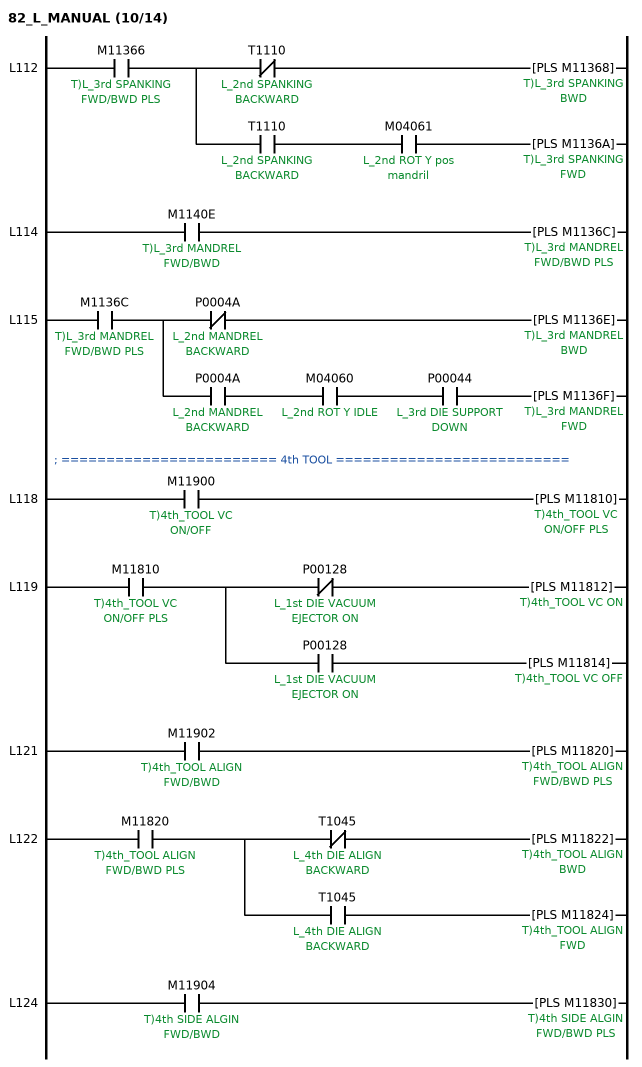
[picture p336: 82_L_MANUAL rungs L112-L124]
; L112
LOAD      M11366	// T)L_3rd SPANKING FWD/BWD PLS
MPUSH
AND NOT   T1110	// L_2nd SPANKING BACKWARD
OUTP      M11368	// T)L_3rd SPANKING BWD
MPOP
AND       T1110	// L_2nd SPANKING BACKWARD
AND       M04061	// L_2nd ROT Y pos mandril
OUTP      M1136A	// T)L_3rd SPANKING FWD
; L114
LOAD      M1140E	// T)L_3rd MANDREL FWD/BWD
OUTP      M1136C	// T)L_3rd MANDREL FWD/BWD PLS
; L115
LOAD      M1136C	// T)L_3rd MANDREL FWD/BWD PLS
MPUSH
AND NOT   P0004A	// L_2nd MANDREL BACKWARD
OUTP      M1136E	// T)L_3rd MANDREL BWD
MPOP
AND       P0004A	// L_2nd MANDREL BACKWARD
AND       M04060	// L_2nd ROT Y IDLE
AND       P00044	// L_3rd DIE SUPPORT DOWN
OUTP      M1136F	// T)L_3rd MANDREL FWD
// ======================== 4th TOOL ==========================
; L118
LOAD      M11900	// T)4th_TOOL VC ON/OFF
OUTP      M11810	// T)4th_TOOL VC ON/OFF PLS
; L119
LOAD      M11810	// T)4th_TOOL VC ON/OFF PLS
MPUSH
AND NOT   P00128	// L_1st DIE VACUUM EJECTOR ON
OUTP      M11812	// T)4th_TOOL VC ON
MPOP
AND       P00128	// L_1st DIE VACUUM EJECTOR ON
OUTP      M11814	// T)4th_TOOL VC OFF
; L121
LOAD      M11902	// T)4th_TOOL ALIGN FWD/BWD
OUTP      M11820	// T)4th_TOOL ALIGN FWD/BWD PLS
; L122
LOAD      M11820	// T)4th_TOOL ALIGN FWD/BWD PLS
MPUSH
AND NOT   T1045	// L_4th DIE ALIGN BACKWARD
OUTP      M11822	// T)4th_TOOL ALIGN BWD
MPOP
AND       T1045	// L_4th DIE ALIGN BACKWARD
OUTP      M11824	// T)4th_TOOL ALIGN FWD
; L124
LOAD      M11904	// T)4th SIDE ALGIN FWD/BWD
OUTP      M11830	// T)4th SIDE ALGIN FWD/BWD PLS

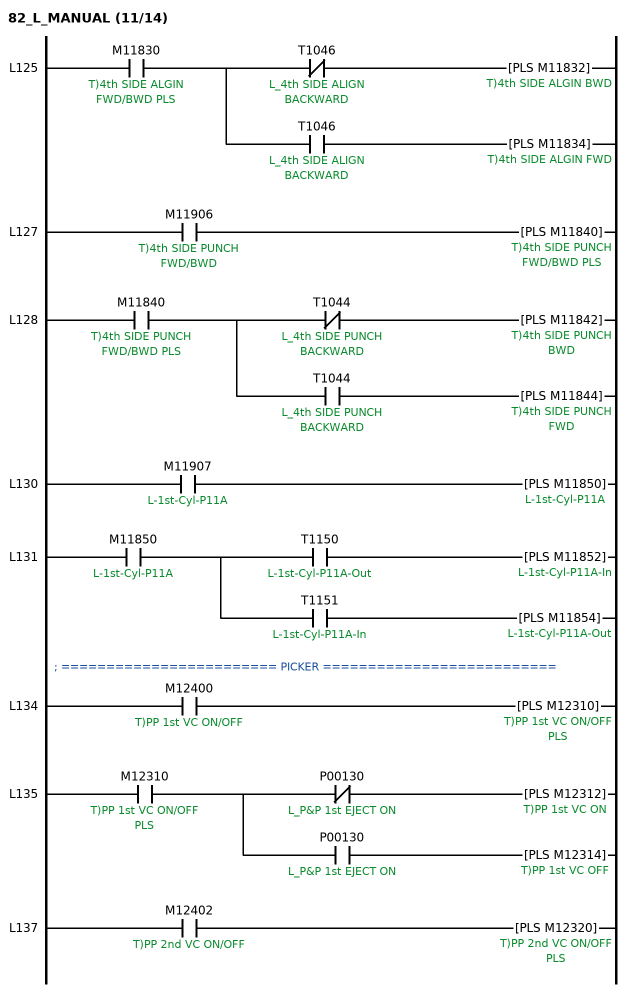
; L125
LOAD      M11830	// T)4th SIDE ALGIN FWD/BWD PLS
MPUSH
AND NOT   T1046	// L_4th SIDE ALIGN BACKWARD
OUTP      M11832	// T)4th SIDE ALGIN BWD
MPOP
AND       T1046	// L_4th SIDE ALIGN BACKWARD
OUTP      M11834	// T)4th SIDE ALGIN FWD
; L127
LOAD      M11906	// T)4th SIDE PUNCH FWD/BWD
OUTP      M11840	// T)4th SIDE PUNCH FWD/BWD PLS
; L128
LOAD      M11840	// T)4th SIDE PUNCH FWD/BWD PLS
MPUSH
AND NOT   T1044	// L_4th SIDE PUNCH BACKWARD
OUTP      M11842	// T)4th SIDE PUNCH BWD
MPOP
AND       T1044	// L_4th SIDE PUNCH BACKWARD
OUTP      M11844	// T)4th SIDE PUNCH FWD
; L130
LOAD      M11907	// L-1st-Cyl-P11A
OUTP      M11850	// L-1st-Cyl-P11A
; L131
LOAD      M11850	// L-1st-Cyl-P11A
MPUSH
AND       T1150	// L-1st-Cyl-P11A-Out
OUTP      M11852	// L-1st-Cyl-P11A-In
MPOP
AND       T1151	// L-1st-Cyl-P11A-In
OUTP      M11854	// L-1st-Cyl-P11A-Out
// ======================== PICKER ==========================
; L134
LOAD      M12400	// T)PP 1st VC ON/OFF
OUTP      M12310	// T)PP 1st VC ON/OFF PLS
; L135
LOAD      M12310	// T)PP 1st VC ON/OFF PLS
MPUSH
AND NOT   P00130	// L_P&P 1st EJECT ON
OUTP      M12312	// T)PP 1st VC ON
MPOP
AND       P00130	// L_P&P 1st EJECT ON
OUTP      M12314	// T)PP 1st VC OFF
; L137
LOAD      M12402	// T)PP 2nd VC ON/OFF
OUTP      M12320	// T)PP 2nd VC ON/OFF PLS

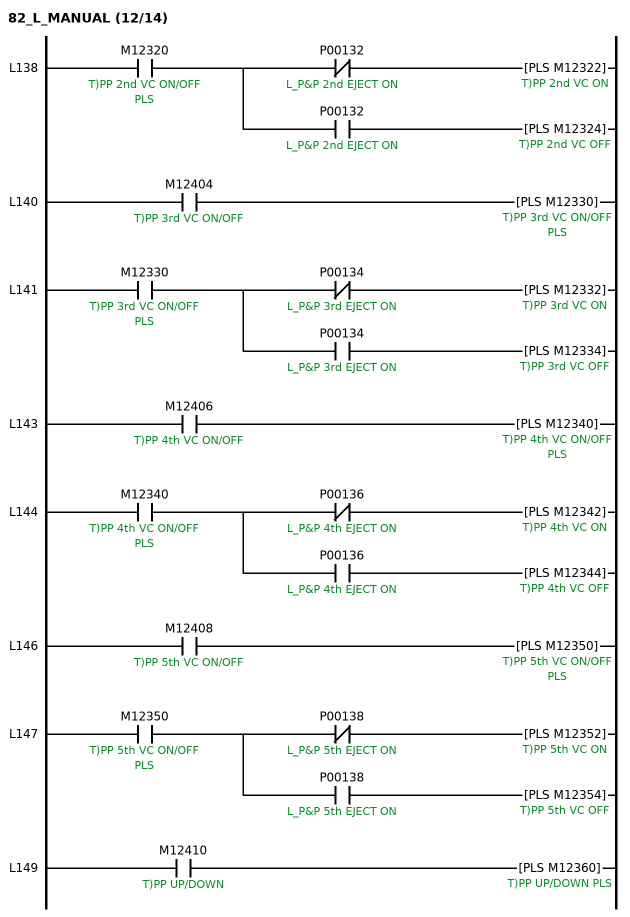
; L138
LOAD      M12320	// T)PP 2nd VC ON/OFF PLS
MPUSH
AND NOT   P00132	// L_P&P 2nd EJECT ON
OUTP      M12322	// T)PP 2nd VC ON
MPOP
AND       P00132	// L_P&P 2nd EJECT ON
OUTP      M12324	// T)PP 2nd VC OFF
; L140
LOAD      M12404	// T)PP 3rd VC ON/OFF
OUTP      M12330	// T)PP 3rd VC ON/OFF PLS
; L141
LOAD      M12330	// T)PP 3rd VC ON/OFF PLS
MPUSH
AND NOT   P00134	// L_P&P 3rd EJECT ON
OUTP      M12332	// T)PP 3rd VC ON
MPOP
AND       P00134	// L_P&P 3rd EJECT ON
OUTP      M12334	// T)PP 3rd VC OFF
; L143
LOAD      M12406	// T)PP 4th VC ON/OFF
OUTP      M12340	// T)PP 4th VC ON/OFF PLS
; L144
LOAD      M12340	// T)PP 4th VC ON/OFF PLS
MPUSH
AND NOT   P00136	// L_P&P 4th EJECT ON
OUTP      M12342	// T)PP 4th VC ON
MPOP
AND       P00136	// L_P&P 4th EJECT ON
OUTP      M12344	// T)PP 4th VC OFF
; L146
LOAD      M12408	// T)PP 5th VC ON/OFF
OUTP      M12350	// T)PP 5th VC ON/OFF PLS
; L147
LOAD      M12350	// T)PP 5th VC ON/OFF PLS
MPUSH
AND NOT   P00138	// L_P&P 5th EJECT ON
OUTP      M12352	// T)PP 5th VC ON
MPOP
AND       P00138	// L_P&P 5th EJECT ON
OUTP      M12354	// T)PP 5th VC OFF
; L149
LOAD      M12410	// T)PP UP/DOWN
OUTP      M12360	// T)PP UP/DOWN PLS

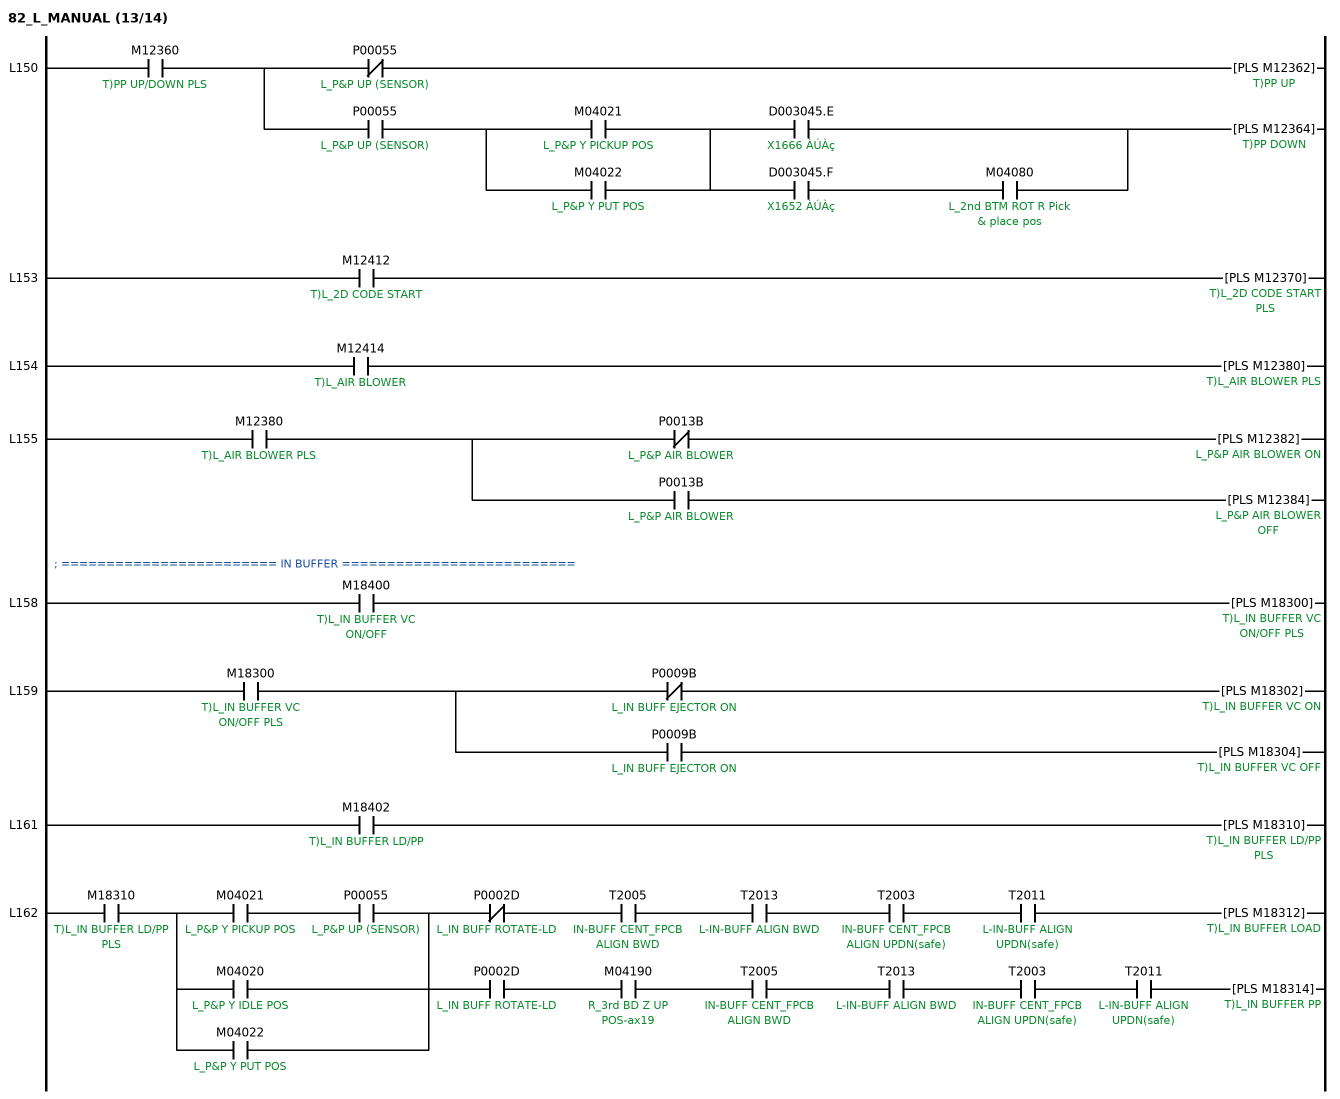
; L150
LOAD      M12360	// T)PP UP/DOWN PLS
MPUSH
AND NOT   P00055	// L_P&P UP (SENSOR)
OUTP      M12362	// T)PP UP
MPOP
AND       P00055	// L_P&P UP (SENSOR)
LOAD      M04021	// L_P&P Y PICKUP POS
OR        M04022	// L_P&P Y PUT POS
AND LOAD
LOAD      D003045.E	// X1666 ÀÚÀç
LOAD      D003045.F	// X1652 ÀÚÀç
AND       M04080	// L_2nd BTM ROT R Pick & place pos
OR LOAD
AND LOAD
OUTP      M12364	// T)PP DOWN
; L153
LOAD      M12412	// T)L_2D CODE START
OUTP      M12370	// T)L_2D CODE START PLS
; L154
LOAD      M12414	// T)L_AIR BLOWER
OUTP      M12380	// T)L_AIR BLOWER PLS
; L155
LOAD      M12380	// T)L_AIR BLOWER PLS
MPUSH
AND NOT   P0013B	// L_P&P AIR BLOWER
OUTP      M12382	// L_P&P AIR BLOWER ON
MPOP
AND       P0013B	// L_P&P AIR BLOWER
OUTP      M12384	// L_P&P AIR BLOWER OFF
// ======================== IN BUFFER ==========================
; L158
LOAD      M18400	// T)L_IN BUFFER VC ON/OFF
OUTP      M18300	// T)L_IN BUFFER VC ON/OFF PLS
; L159
LOAD      M18300	// T)L_IN BUFFER VC ON/OFF PLS
MPUSH
AND NOT   P0009B	// L_IN BUFF EJECTOR ON
OUTP      M18302	// T)L_IN BUFFER VC ON
MPOP
AND       P0009B	// L_IN BUFF EJECTOR ON
OUTP      M18304	// T)L_IN BUFFER VC OFF
; L161
LOAD      M18402	// T)L_IN BUFFER LD/PP
OUTP      M18310	// T)L_IN BUFFER LD/PP PLS
; L162
LOAD      M18310	// T)L_IN BUFFER LD/PP PLS
LOAD      M04021	// L_P&P Y PICKUP POS
AND       P00055	// L_P&P UP (SENSOR)
OR        M04020	// L_P&P Y IDLE POS
OR        M04022	// L_P&P Y PUT POS
AND LOAD
MPUSH
AND NOT   P0002D	// L_IN BUFF ROTATE-LD
AND       T2005	// IN-BUFF CENT_FPCB ALIGN BWD
AND       T2013	// L-IN-BUFF ALIGN BWD
AND       T2003	// IN-BUFF CENT_FPCB ALIGN UPDN(safe)
AND       T2011	// L-IN-BUFF ALIGN UPDN(safe)
OUTP      M18312	// T)L_IN BUFFER LOAD
MPOP
AND       P0002D	// L_IN BUFF ROTATE-LD
AND       M04190	// R_3rd BD Z UP POS-ax19
AND       T2005	// IN-BUFF CENT_FPCB ALIGN BWD
AND       T2013	// L-IN-BUFF ALIGN BWD
AND       T2003	// IN-BUFF CENT_FPCB ALIGN UPDN(safe)
AND       T2011	// L-IN-BUFF ALIGN UPDN(safe)
OUTP      M18314	// T)L_IN BUFFER PP

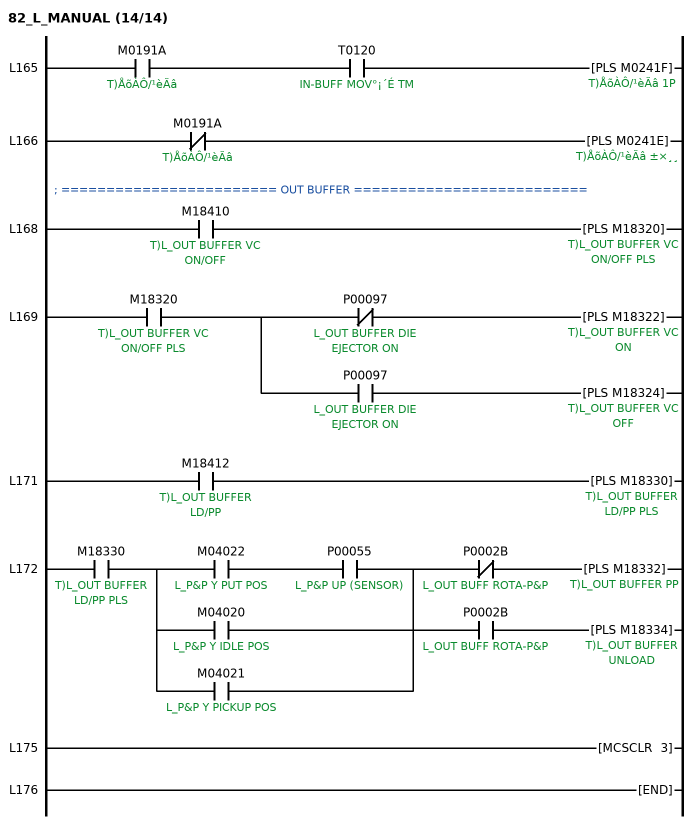
; L165
LOAD      M0191A	// T)ÅõÀÔ/¹èÃâ
AND       T0120	// IN-BUFF MOV°¡´É TM
OUTP      M0241F	// T)ÅõÀÔ/¹èÃâ 1P
; L166
LOAD NOT  M0191A	// T)ÅõÀÔ/¹èÃâ
OUTP      M0241E	// T)ÅõÀÔ/¹èÃâ ±×¸¸
// ======================== OUT BUFFER ==========================
; L168
LOAD      M18410	// T)L_OUT BUFFER VC ON/OFF
OUTP      M18320	// T)L_OUT BUFFER VC ON/OFF PLS
; L169
LOAD      M18320	// T)L_OUT BUFFER VC ON/OFF PLS
MPUSH
AND NOT   P00097	// L_OUT BUFFER DIE EJECTOR ON
OUTP      M18322	// T)L_OUT BUFFER VC ON
MPOP
AND       P00097	// L_OUT BUFFER DIE EJECTOR ON
OUTP      M18324	// T)L_OUT BUFFER VC OFF
; L171
LOAD      M18412	// T)L_OUT BUFFER LD/PP
OUTP      M18330	// T)L_OUT BUFFER LD/PP PLS
; L172
LOAD      M18330	// T)L_OUT BUFFER LD/PP PLS
LOAD      M04022	// L_P&P Y PUT POS
AND       P00055	// L_P&P UP (SENSOR)
OR        M04020	// L_P&P Y IDLE POS
OR        M04021	// L_P&P Y PICKUP POS
AND LOAD
MPUSH
AND NOT   P0002B	// L_OUT BUFF ROTA-P&P
OUTP      M18332	// T)L_OUT BUFFER PP
MPOP
AND       P0002B	// L_OUT BUFF ROTA-P&P
OUTP      M18334	// T)L_OUT BUFFER UNLOAD
; L175
MCSCLR    3
; L176
END

PROGRAM 83_R_MANUAL (task: ½ºÄµ ÇÁ·Î±×·¥)

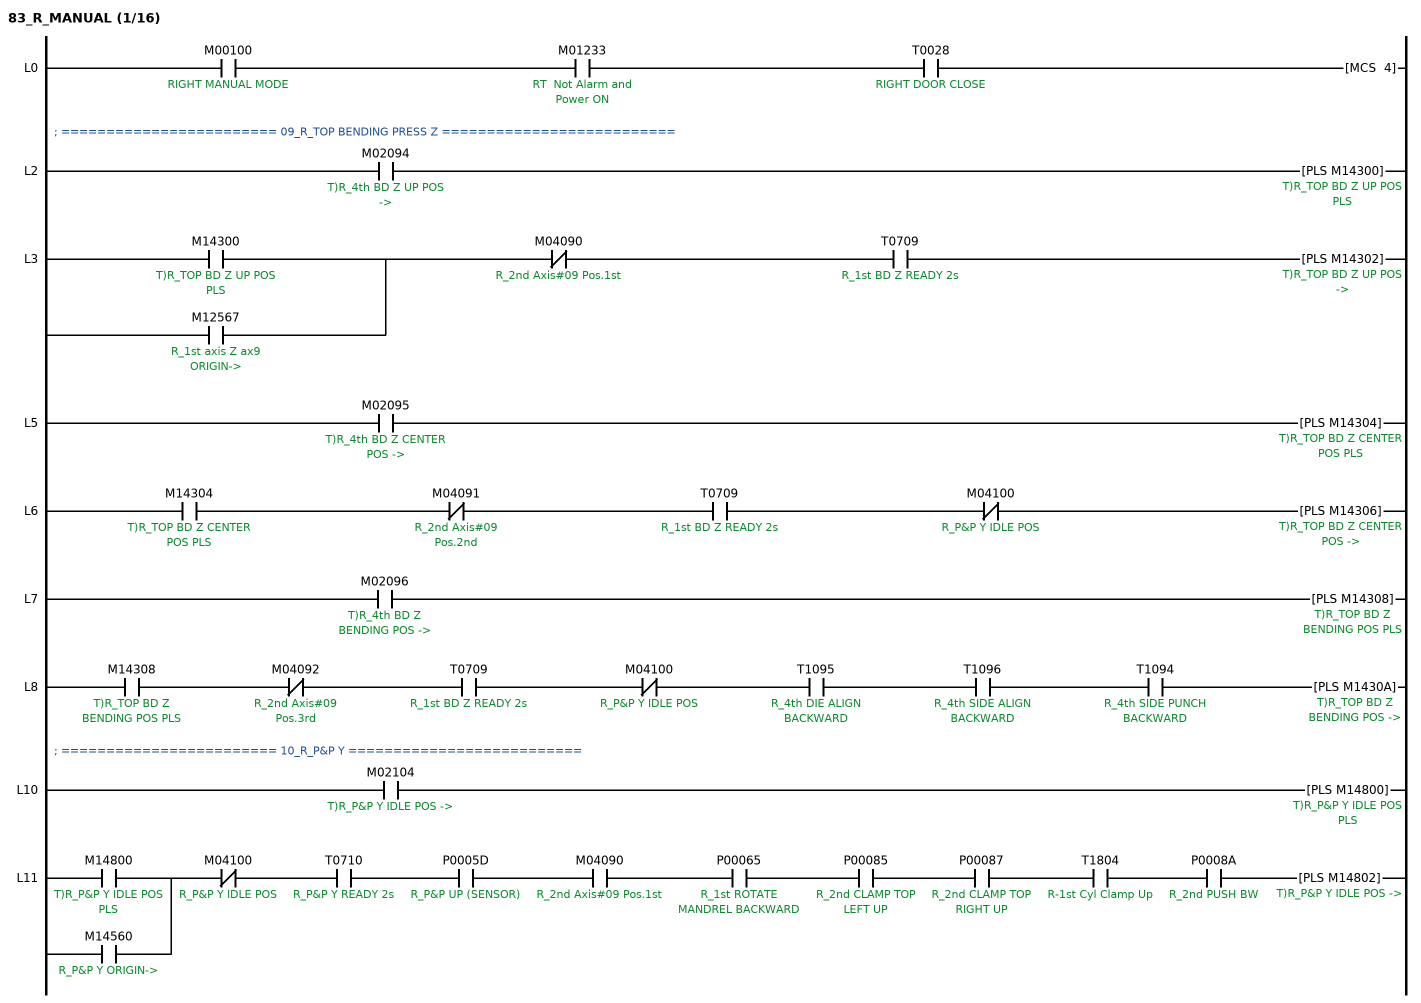
; L0
LOAD      M00100	// RIGHT MANUAL MODE
AND       M01233	// RT  Not Alarm and Power ON
AND       T0028	// RIGHT DOOR CLOSE
MCS       4
// ======================== 09_R_TOP BENDING PRESS Z ==========================
; L2
LOAD      M02094	// T)R_4th BD Z UP POS ->
OUTP      M14300	// T)R_TOP BD Z UP POS PLS
; L3
LOAD      M14300	// T)R_TOP BD Z UP POS PLS
OR        M12567	// R_1st axis Z ax9 ORIGIN->
AND NOT   M04090	// R_2nd Axis#09 Pos.1st
AND       T0709	// R_1st BD Z READY 2s
OUTP      M14302	// T)R_TOP BD Z UP POS ->
; L5
LOAD      M02095	// T)R_4th BD Z CENTER POS ->
OUTP      M14304	// T)R_TOP BD Z CENTER POS PLS
; L6
LOAD      M14304	// T)R_TOP BD Z CENTER POS PLS
AND NOT   M04091	// R_2nd Axis#09 Pos.2nd
AND       T0709	// R_1st BD Z READY 2s
AND NOT   M04100	// R_P&P Y IDLE POS
OUTP      M14306	// T)R_TOP BD Z CENTER POS ->
; L7
LOAD      M02096	// T)R_4th BD Z BENDING POS ->
OUTP      M14308	// T)R_TOP BD Z BENDING POS PLS
; L8
LOAD      M14308	// T)R_TOP BD Z BENDING POS PLS
AND NOT   M04092	// R_2nd Axis#09 Pos.3rd
AND       T0709	// R_1st BD Z READY 2s
AND NOT   M04100	// R_P&P Y IDLE POS
AND       T1095	// R_4th DIE ALIGN BACKWARD
AND       T1096	// R_4th SIDE ALIGN BACKWARD
AND       T1094	// R_4th SIDE PUNCH BACKWARD
OUTP      M1430A	// T)R_TOP BD Z BENDING POS ->
// ======================== 10_R_P&P Y ==========================
; L10
LOAD      M02104	// T)R_P&P Y IDLE POS ->
OUTP      M14800	// T)R_P&P Y IDLE POS PLS
; L11
LOAD      M14800	// T)R_P&P Y IDLE POS PLS
OR        M14560	// R_P&P Y ORIGIN->
AND NOT   M04100	// R_P&P Y IDLE POS
AND       T0710	// R_P&P Y READY 2s
AND       P0005D	// R_P&P UP (SENSOR)
AND       M04090	// R_2nd Axis#09 Pos.1st
AND       P00065	// R_1st ROTATE MANDREL BACKWARD
AND       P00085	// R_2nd CLAMP TOP LEFT UP
AND       P00087	// R_2nd CLAMP TOP RIGHT UP
AND       T1804	// R-1st Cyl Clamp Up
AND       P0008A	// R_2nd PUSH BW
OUTP      M14802	// T)R_P&P Y IDLE POS ->

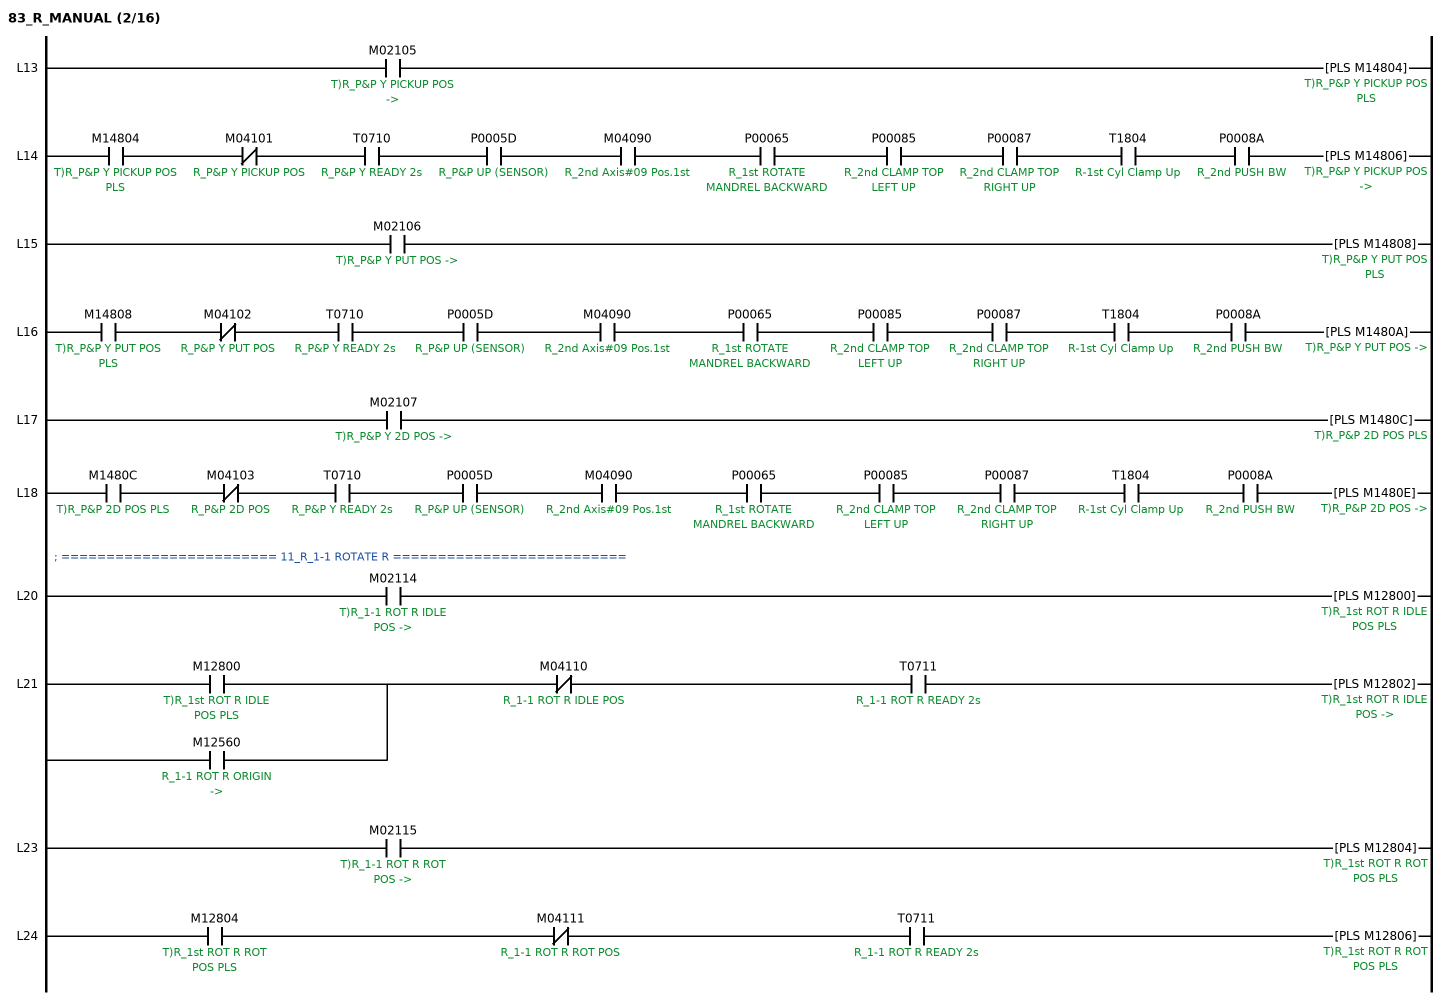
; L13
LOAD      M02105	// T)R_P&P Y PICKUP POS ->
OUTP      M14804	// T)R_P&P Y PICKUP POS PLS
; L14
LOAD      M14804	// T)R_P&P Y PICKUP POS PLS
AND NOT   M04101	// R_P&P Y PICKUP POS
AND       T0710	// R_P&P Y READY 2s
AND       P0005D	// R_P&P UP (SENSOR)
AND       M04090	// R_2nd Axis#09 Pos.1st
AND       P00065	// R_1st ROTATE MANDREL BACKWARD
AND       P00085	// R_2nd CLAMP TOP LEFT UP
AND       P00087	// R_2nd CLAMP TOP RIGHT UP
AND       T1804	// R-1st Cyl Clamp Up
AND       P0008A	// R_2nd PUSH BW
OUTP      M14806	// T)R_P&P Y PICKUP POS ->
; L15
LOAD      M02106	// T)R_P&P Y PUT POS ->
OUTP      M14808	// T)R_P&P Y PUT POS PLS
; L16
LOAD      M14808	// T)R_P&P Y PUT POS PLS
AND NOT   M04102	// R_P&P Y PUT POS
AND       T0710	// R_P&P Y READY 2s
AND       P0005D	// R_P&P UP (SENSOR)
AND       M04090	// R_2nd Axis#09 Pos.1st
AND       P00065	// R_1st ROTATE MANDREL BACKWARD
AND       P00085	// R_2nd CLAMP TOP LEFT UP
AND       P00087	// R_2nd CLAMP TOP RIGHT UP
AND       T1804	// R-1st Cyl Clamp Up
AND       P0008A	// R_2nd PUSH BW
OUTP      M1480A	// T)R_P&P Y PUT POS ->
; L17
LOAD      M02107	// T)R_P&P Y 2D POS ->
OUTP      M1480C	// T)R_P&P 2D POS PLS
; L18
LOAD      M1480C	// T)R_P&P 2D POS PLS
AND NOT   M04103	// R_P&P 2D POS
AND       T0710	// R_P&P Y READY 2s
AND       P0005D	// R_P&P UP (SENSOR)
AND       M04090	// R_2nd Axis#09 Pos.1st
AND       P00065	// R_1st ROTATE MANDREL BACKWARD
AND       P00085	// R_2nd CLAMP TOP LEFT UP
AND       P00087	// R_2nd CLAMP TOP RIGHT UP
AND       T1804	// R-1st Cyl Clamp Up
AND       P0008A	// R_2nd PUSH BW
OUTP      M1480E	// T)R_P&P 2D POS ->
// ======================== 11_R_1-1 ROTATE R ==========================
; L20
LOAD      M02114	// T)R_1-1 ROT R IDLE POS ->
OUTP      M12800	// T)R_1st ROT R IDLE POS PLS
; L21
LOAD      M12800	// T)R_1st ROT R IDLE POS PLS
OR        M12560	// R_1-1 ROT R ORIGIN ->
AND NOT   M04110	// R_1-1 ROT R IDLE POS
AND       T0711	// R_1-1 ROT R READY 2s
OUTP      M12802	// T)R_1st ROT R IDLE POS ->
; L23
LOAD      M02115	// T)R_1-1 ROT R ROT POS ->
OUTP      M12804	// T)R_1st ROT R ROT POS PLS
; L24
LOAD      M12804	// T)R_1st ROT R ROT POS PLS
AND NOT   M04111	// R_1-1 ROT R ROT POS
AND       T0711	// R_1-1 ROT R READY 2s
OUTP      M12806	// T)R_1st ROT R ROT POS PLS

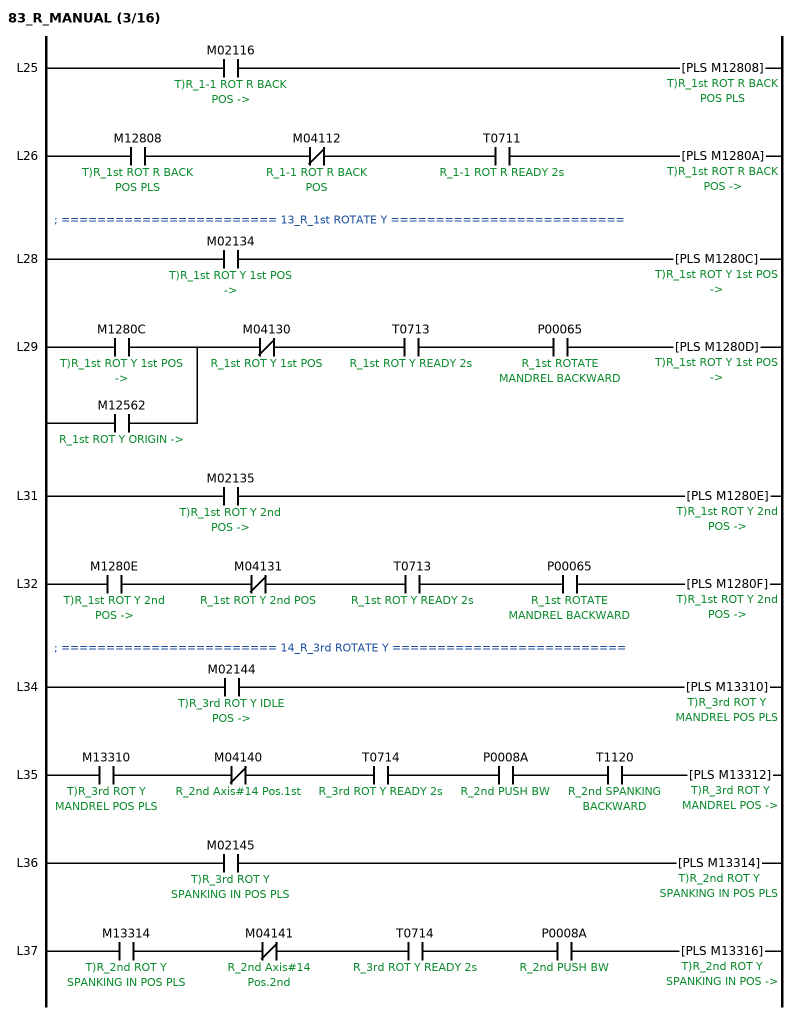
; L25
LOAD      M02116	// T)R_1-1 ROT R BACK POS ->
OUTP      M12808	// T)R_1st ROT R BACK POS PLS
; L26
LOAD      M12808	// T)R_1st ROT R BACK POS PLS
AND NOT   M04112	// R_1-1 ROT R BACK POS
AND       T0711	// R_1-1 ROT R READY 2s
OUTP      M1280A	// T)R_1st ROT R BACK POS ->
// ======================== 13_R_1st ROTATE Y ==========================
; L28
LOAD      M02134	// T)R_1st ROT Y 1st POS ->
OUTP      M1280C	// T)R_1st ROT Y 1st POS ->
; L29
LOAD      M1280C	// T)R_1st ROT Y 1st POS ->
OR        M12562	// R_1st ROT Y ORIGIN ->
AND NOT   M04130	// R_1st ROT Y 1st POS
AND       T0713	// R_1st ROT Y READY 2s
AND       P00065	// R_1st ROTATE MANDREL BACKWARD
OUTP      M1280D	// T)R_1st ROT Y 1st POS ->
; L31
LOAD      M02135	// T)R_1st ROT Y 2nd POS ->
OUTP      M1280E	// T)R_1st ROT Y 2nd POS ->
; L32
LOAD      M1280E	// T)R_1st ROT Y 2nd POS ->
AND NOT   M04131	// R_1st ROT Y 2nd POS
AND       T0713	// R_1st ROT Y READY 2s
AND       P00065	// R_1st ROTATE MANDREL BACKWARD
OUTP      M1280F	// T)R_1st ROT Y 2nd POS ->
// ======================== 14_R_3rd ROTATE Y ==========================
; L34
LOAD      M02144	// T)R_3rd ROT Y IDLE POS ->
OUTP      M13310	// T)R_3rd ROT Y MANDREL POS PLS
; L35
LOAD      M13310	// T)R_3rd ROT Y MANDREL POS PLS
AND NOT   M04140	// R_2nd Axis#14 Pos.1st
AND       T0714	// R_3rd ROT Y READY 2s
AND       P0008A	// R_2nd PUSH BW
AND       T1120	// R_2nd SPANKING BACKWARD
OUTP      M13312	// T)R_3rd ROT Y MANDREL POS ->
; L36
LOAD      M02145	// T)R_3rd ROT Y SPANKING IN POS PLS
OUTP      M13314	// T)R_2nd ROT Y SPANKING IN POS PLS
; L37
LOAD      M13314	// T)R_2nd ROT Y SPANKING IN POS PLS
AND NOT   M04141	// R_2nd Axis#14 Pos.2nd
AND       T0714	// R_3rd ROT Y READY 2s
AND       P0008A	// R_2nd PUSH BW
OUTP      M13316	// T)R_2nd ROT Y SPANKING IN POS ->

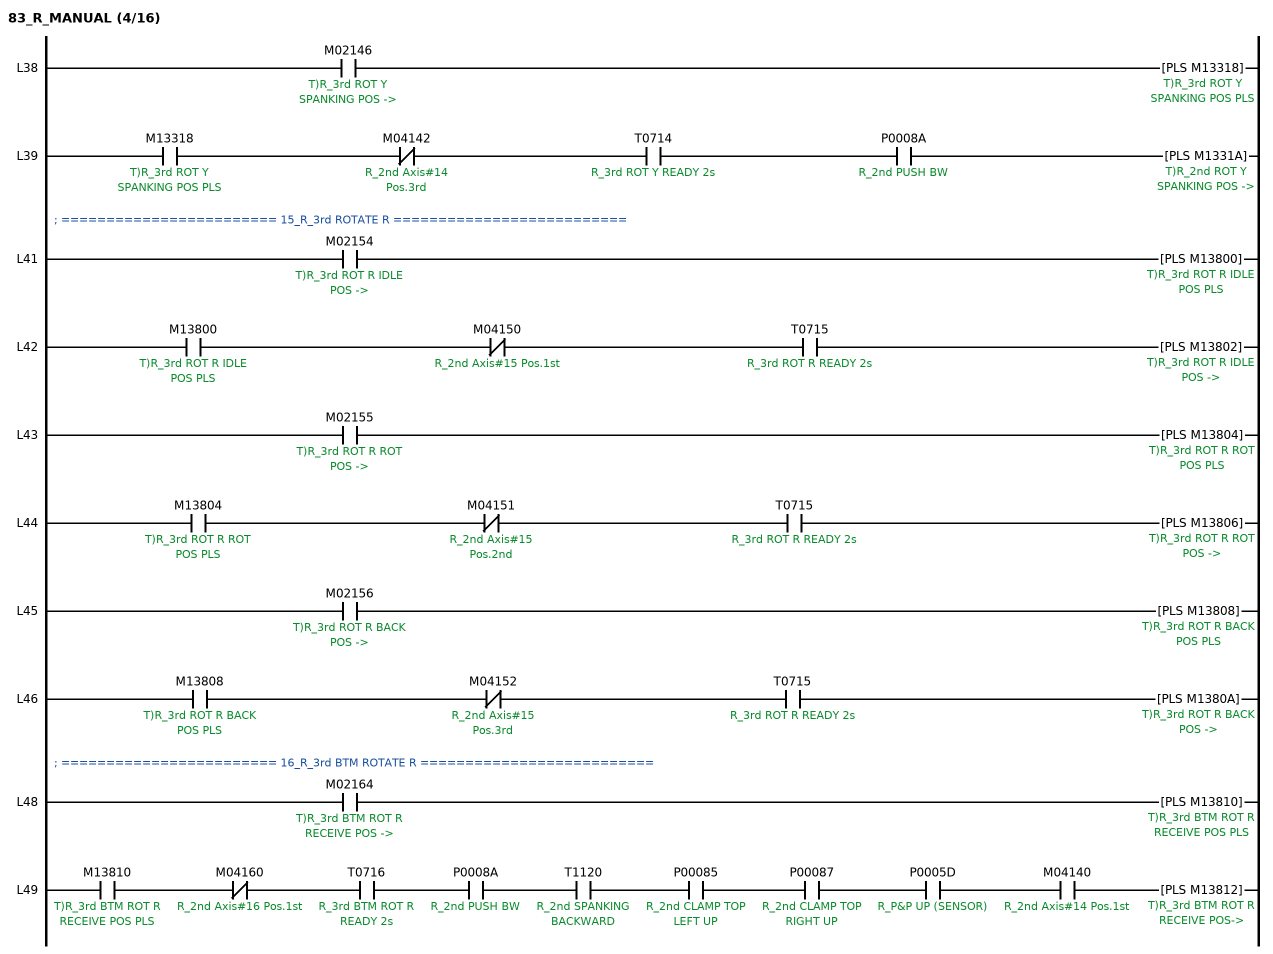
; L38
LOAD      M02146	// T)R_3rd ROT Y SPANKING POS ->
OUTP      M13318	// T)R_3rd ROT Y SPANKING POS PLS
; L39
LOAD      M13318	// T)R_3rd ROT Y SPANKING POS PLS
AND NOT   M04142	// R_2nd Axis#14 Pos.3rd
AND       T0714	// R_3rd ROT Y READY 2s
AND       P0008A	// R_2nd PUSH BW
OUTP      M1331A	// T)R_2nd ROT Y SPANKING POS ->
// ======================== 15_R_3rd ROTATE R ==========================
; L41
LOAD      M02154	// T)R_3rd ROT R IDLE POS ->
OUTP      M13800	// T)R_3rd ROT R IDLE POS PLS
; L42
LOAD      M13800	// T)R_3rd ROT R IDLE POS PLS
AND NOT   M04150	// R_2nd Axis#15 Pos.1st
AND       T0715	// R_3rd ROT R READY 2s
OUTP      M13802	// T)R_3rd ROT R IDLE POS ->
; L43
LOAD      M02155	// T)R_3rd ROT R ROT POS ->
OUTP      M13804	// T)R_3rd ROT R ROT POS PLS
; L44
LOAD      M13804	// T)R_3rd ROT R ROT POS PLS
AND NOT   M04151	// R_2nd Axis#15 Pos.2nd
AND       T0715	// R_3rd ROT R READY 2s
OUTP      M13806	// T)R_3rd ROT R ROT POS ->
; L45
LOAD      M02156	// T)R_3rd ROT R BACK POS ->
OUTP      M13808	// T)R_3rd ROT R BACK POS PLS
; L46
LOAD      M13808	// T)R_3rd ROT R BACK POS PLS
AND NOT   M04152	// R_2nd Axis#15 Pos.3rd
AND       T0715	// R_3rd ROT R READY 2s
OUTP      M1380A	// T)R_3rd ROT R BACK POS ->
// ======================== 16_R_3rd BTM ROTATE R ==========================
; L48
LOAD      M02164	// T)R_3rd BTM ROT R RECEIVE POS ->
OUTP      M13810	// T)R_3rd BTM ROT R RECEIVE POS PLS
; L49
LOAD      M13810	// T)R_3rd BTM ROT R RECEIVE POS PLS
AND NOT   M04160	// R_2nd Axis#16 Pos.1st
AND       T0716	// R_3rd BTM ROT R READY 2s
AND       P0008A	// R_2nd PUSH BW
AND       T1120	// R_2nd SPANKING BACKWARD
AND       P00085	// R_2nd CLAMP TOP LEFT UP
AND       P00087	// R_2nd CLAMP TOP RIGHT UP
AND       P0005D	// R_P&P UP (SENSOR)
AND       M04140	// R_2nd Axis#14 Pos.1st
OUTP      M13812	// T)R_3rd BTM ROT R RECEIVE POS->

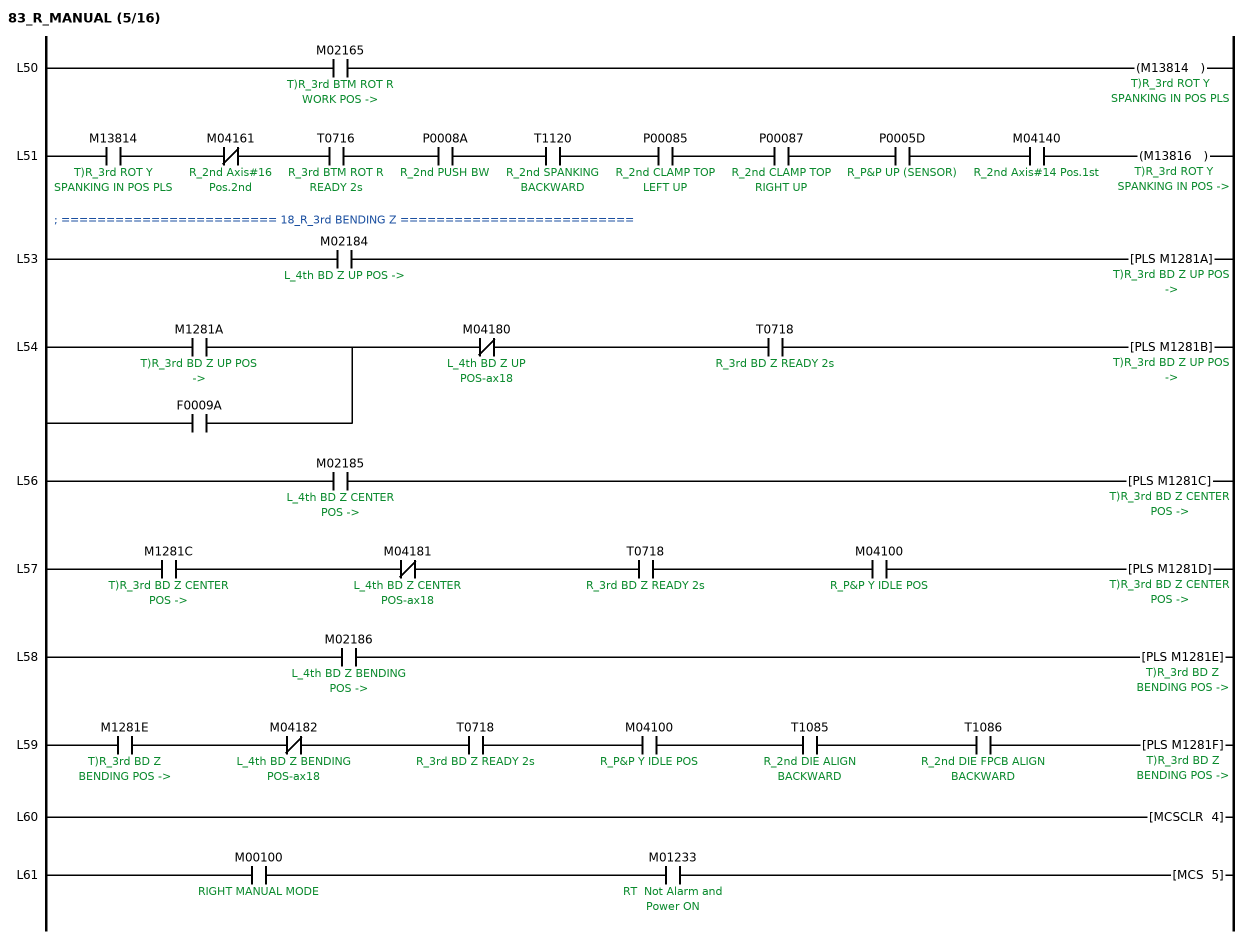
; L50
LOAD      M02165	// T)R_3rd BTM ROT R WORK POS ->
OUT       M13814	// T)R_3rd ROT Y SPANKING IN POS PLS
; L51
LOAD      M13814	// T)R_3rd ROT Y SPANKING IN POS PLS
AND NOT   M04161	// R_2nd Axis#16 Pos.2nd
AND       T0716	// R_3rd BTM ROT R READY 2s
AND       P0008A	// R_2nd PUSH BW
AND       T1120	// R_2nd SPANKING BACKWARD
AND       P00085	// R_2nd CLAMP TOP LEFT UP
AND       P00087	// R_2nd CLAMP TOP RIGHT UP
AND       P0005D	// R_P&P UP (SENSOR)
AND       M04140	// R_2nd Axis#14 Pos.1st
OUT       M13816	// T)R_3rd ROT Y SPANKING IN POS ->
// ======================== 18_R_3rd BENDING Z ==========================
; L53
LOAD      M02184	// L_4th BD Z UP POS ->
OUTP      M1281A	// T)R_3rd BD Z UP POS ->
; L54
LOAD      M1281A	// T)R_3rd BD Z UP POS ->
OR        F0009A
AND NOT   M04180	// L_4th BD Z UP POS-ax18
AND       T0718	// R_3rd BD Z READY 2s
OUTP      M1281B	// T)R_3rd BD Z UP POS ->
; L56
LOAD      M02185	// L_4th BD Z CENTER POS ->
OUTP      M1281C	// T)R_3rd BD Z CENTER POS ->
; L57
LOAD      M1281C	// T)R_3rd BD Z CENTER POS ->
AND NOT   M04181	// L_4th BD Z CENTER POS-ax18
AND       T0718	// R_3rd BD Z READY 2s
AND       M04100	// R_P&P Y IDLE POS
OUTP      M1281D	// T)R_3rd BD Z CENTER POS ->
; L58
LOAD      M02186	// L_4th BD Z BENDING POS ->
OUTP      M1281E	// T)R_3rd BD Z BENDING POS ->
; L59
LOAD      M1281E	// T)R_3rd BD Z BENDING POS ->
AND NOT   M04182	// L_4th BD Z BENDING POS-ax18
AND       T0718	// R_3rd BD Z READY 2s
AND       M04100	// R_P&P Y IDLE POS
AND       T1085	// R_2nd DIE ALIGN BACKWARD
AND       T1086	// R_2nd DIE FPCB ALIGN BACKWARD
OUTP      M1281F	// T)R_3rd BD Z BENDING POS ->
; L60
MCSCLR    4
; L61
LOAD      M00100	// RIGHT MANUAL MODE
AND       M01233	// RT  Not Alarm and Power ON
MCS       5

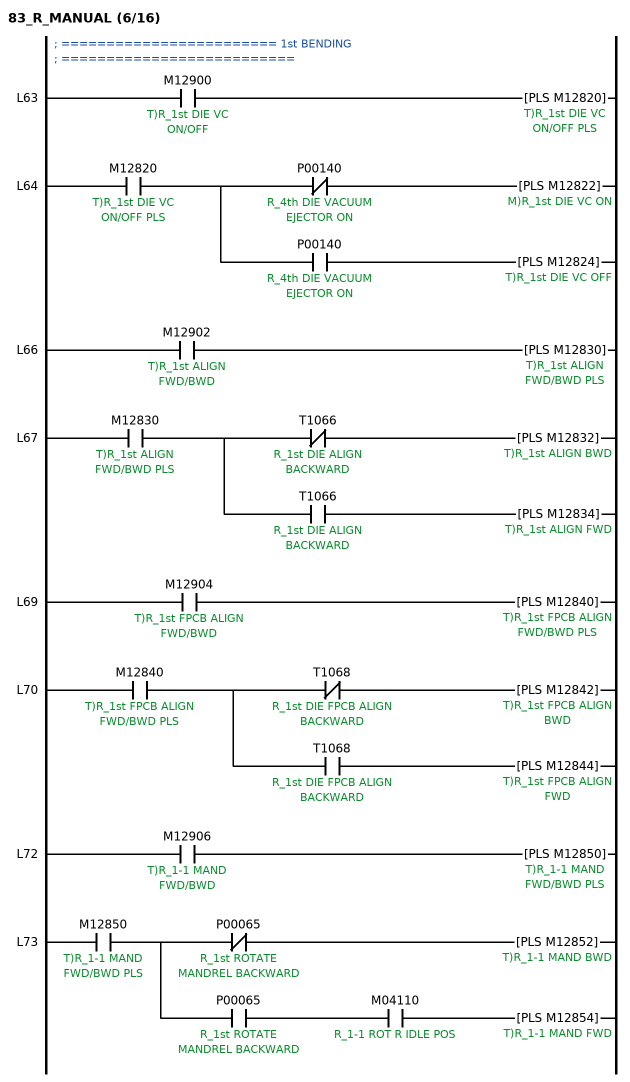
// ======================== 1st BENDING ==========================
; L63
LOAD      M12900	// T)R_1st DIE VC ON/OFF
OUTP      M12820	// T)R_1st DIE VC ON/OFF PLS
; L64
LOAD      M12820	// T)R_1st DIE VC ON/OFF PLS
MPUSH
AND NOT   P00140	// R_4th DIE VACUUM EJECTOR ON
OUTP      M12822	// M)R_1st DIE VC ON
MPOP
AND       P00140	// R_4th DIE VACUUM EJECTOR ON
OUTP      M12824	// T)R_1st DIE VC OFF
; L66
LOAD      M12902	// T)R_1st ALIGN FWD/BWD
OUTP      M12830	// T)R_1st ALIGN FWD/BWD PLS
; L67
LOAD      M12830	// T)R_1st ALIGN FWD/BWD PLS
MPUSH
AND NOT   T1066	// R_1st DIE ALIGN BACKWARD
OUTP      M12832	// T)R_1st ALIGN BWD
MPOP
AND       T1066	// R_1st DIE ALIGN BACKWARD
OUTP      M12834	// T)R_1st ALIGN FWD
; L69
LOAD      M12904	// T)R_1st FPCB ALIGN FWD/BWD
OUTP      M12840	// T)R_1st FPCB ALIGN FWD/BWD PLS
; L70
LOAD      M12840	// T)R_1st FPCB ALIGN FWD/BWD PLS
MPUSH
AND NOT   T1068	// R_1st DIE FPCB ALIGN BACKWARD
OUTP      M12842	// T)R_1st FPCB ALIGN BWD
MPOP
AND       T1068	// R_1st DIE FPCB ALIGN BACKWARD
OUTP      M12844	// T)R_1st FPCB ALIGN FWD
; L72
LOAD      M12906	// T)R_1-1 MAND FWD/BWD
OUTP      M12850	// T)R_1-1 MAND FWD/BWD PLS
; L73
LOAD      M12850	// T)R_1-1 MAND FWD/BWD PLS
MPUSH
AND NOT   P00065	// R_1st ROTATE MANDREL BACKWARD
OUTP      M12852	// T)R_1-1 MAND BWD
MPOP
AND       P00065	// R_1st ROTATE MANDREL BACKWARD
AND       M04110	// R_1-1 ROT R IDLE POS
OUTP      M12854	// T)R_1-1 MAND FWD

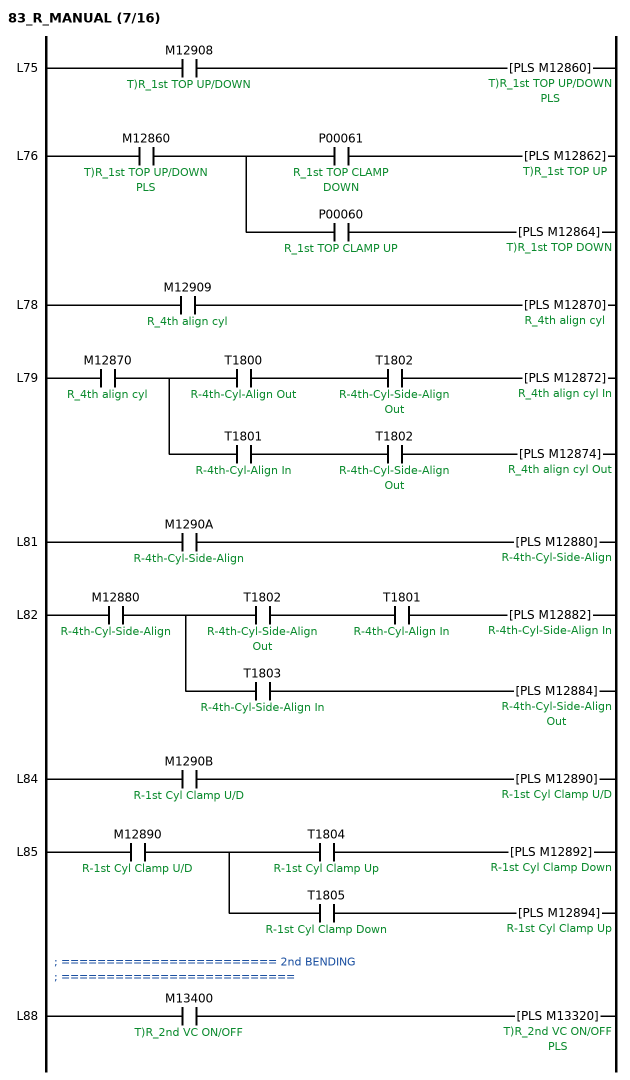
; L75
LOAD      M12908	// T)R_1st TOP UP/DOWN
OUTP      M12860	// T)R_1st TOP UP/DOWN PLS
; L76
LOAD      M12860	// T)R_1st TOP UP/DOWN PLS
MPUSH
AND       P00061	// R_1st TOP CLAMP DOWN
OUTP      M12862	// T)R_1st TOP UP
MPOP
AND       P00060	// R_1st TOP CLAMP UP
OUTP      M12864	// T)R_1st TOP DOWN
; L78
LOAD      M12909	// R_4th align cyl
OUTP      M12870	// R_4th align cyl
; L79
LOAD      M12870	// R_4th align cyl
MPUSH
AND       T1800	// R-4th-Cyl-Align Out
AND       T1802	// R-4th-Cyl-Side-Align Out
OUTP      M12872	// R_4th align cyl In
MPOP
AND       T1801	// R-4th-Cyl-Align In
AND       T1802	// R-4th-Cyl-Side-Align Out
OUTP      M12874	// R_4th align cyl Out
; L81
LOAD      M1290A	// R-4th-Cyl-Side-Align
OUTP      M12880	// R-4th-Cyl-Side-Align
; L82
LOAD      M12880	// R-4th-Cyl-Side-Align
MPUSH
AND       T1802	// R-4th-Cyl-Side-Align Out
AND       T1801	// R-4th-Cyl-Align In
OUTP      M12882	// R-4th-Cyl-Side-Align In
MPOP
AND       T1803	// R-4th-Cyl-Side-Align In
OUTP      M12884	// R-4th-Cyl-Side-Align Out
; L84
LOAD      M1290B	// R-1st Cyl Clamp U/D
OUTP      M12890	// R-1st Cyl Clamp U/D
; L85
LOAD      M12890	// R-1st Cyl Clamp U/D
MPUSH
AND       T1804	// R-1st Cyl Clamp Up
OUTP      M12892	// R-1st Cyl Clamp Down
MPOP
AND       T1805	// R-1st Cyl Clamp Down
OUTP      M12894	// R-1st Cyl Clamp Up
// ======================== 2nd BENDING ==========================
; L88
LOAD      M13400	// T)R_2nd VC ON/OFF
OUTP      M13320	// T)R_2nd VC ON/OFF PLS

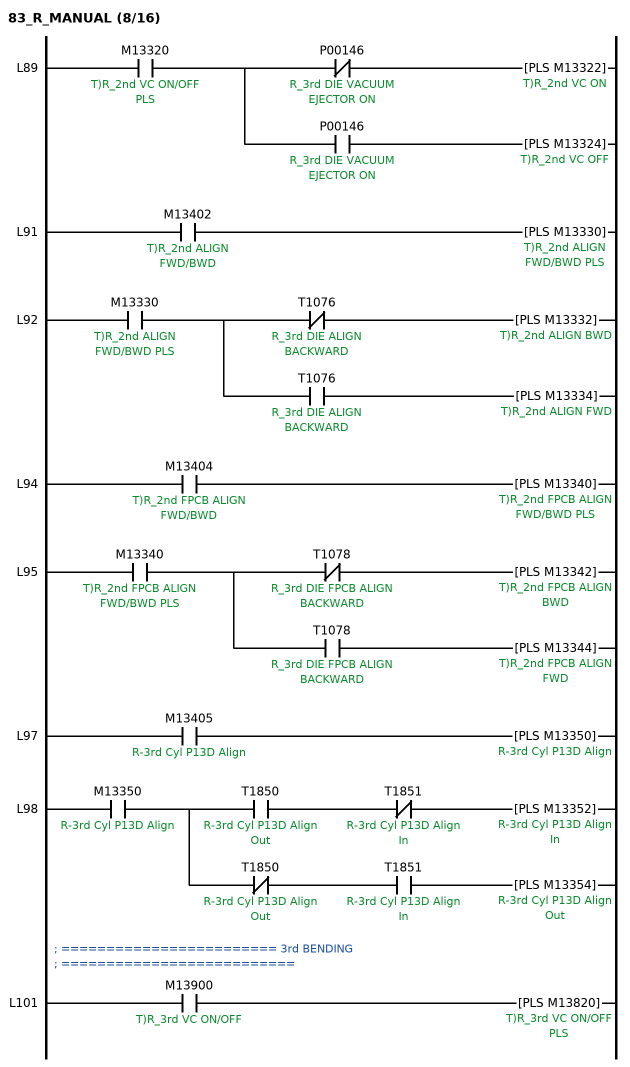
; L89
LOAD      M13320	// T)R_2nd VC ON/OFF PLS
MPUSH
AND NOT   P00146	// R_3rd DIE VACUUM EJECTOR ON
OUTP      M13322	// T)R_2nd VC ON
MPOP
AND       P00146	// R_3rd DIE VACUUM EJECTOR ON
OUTP      M13324	// T)R_2nd VC OFF
; L91
LOAD      M13402	// T)R_2nd ALIGN FWD/BWD
OUTP      M13330	// T)R_2nd ALIGN FWD/BWD PLS
; L92
LOAD      M13330	// T)R_2nd ALIGN FWD/BWD PLS
MPUSH
AND NOT   T1076	// R_3rd DIE ALIGN BACKWARD
OUTP      M13332	// T)R_2nd ALIGN BWD
MPOP
AND       T1076	// R_3rd DIE ALIGN BACKWARD
OUTP      M13334	// T)R_2nd ALIGN FWD
; L94
LOAD      M13404	// T)R_2nd FPCB ALIGN FWD/BWD
OUTP      M13340	// T)R_2nd FPCB ALIGN FWD/BWD PLS
; L95
LOAD      M13340	// T)R_2nd FPCB ALIGN FWD/BWD PLS
MPUSH
AND NOT   T1078	// R_3rd DIE FPCB ALIGN BACKWARD
OUTP      M13342	// T)R_2nd FPCB ALIGN BWD
MPOP
AND       T1078	// R_3rd DIE FPCB ALIGN BACKWARD
OUTP      M13344	// T)R_2nd FPCB ALIGN FWD
; L97
LOAD      M13405	// R-3rd Cyl P13D Align
OUTP      M13350	// R-3rd Cyl P13D Align
; L98
LOAD      M13350	// R-3rd Cyl P13D Align
MPUSH
AND       T1850	// R-3rd Cyl P13D Align Out
AND NOT   T1851	// R-3rd Cyl P13D Align In
OUTP      M13352	// R-3rd Cyl P13D Align In
MPOP
AND NOT   T1850	// R-3rd Cyl P13D Align Out
AND       T1851	// R-3rd Cyl P13D Align In
OUTP      M13354	// R-3rd Cyl P13D Align Out
// ======================== 3rd BENDING ==========================
; L101
LOAD      M13900	// T)R_3rd VC ON/OFF
OUTP      M13820	// T)R_3rd VC ON/OFF PLS

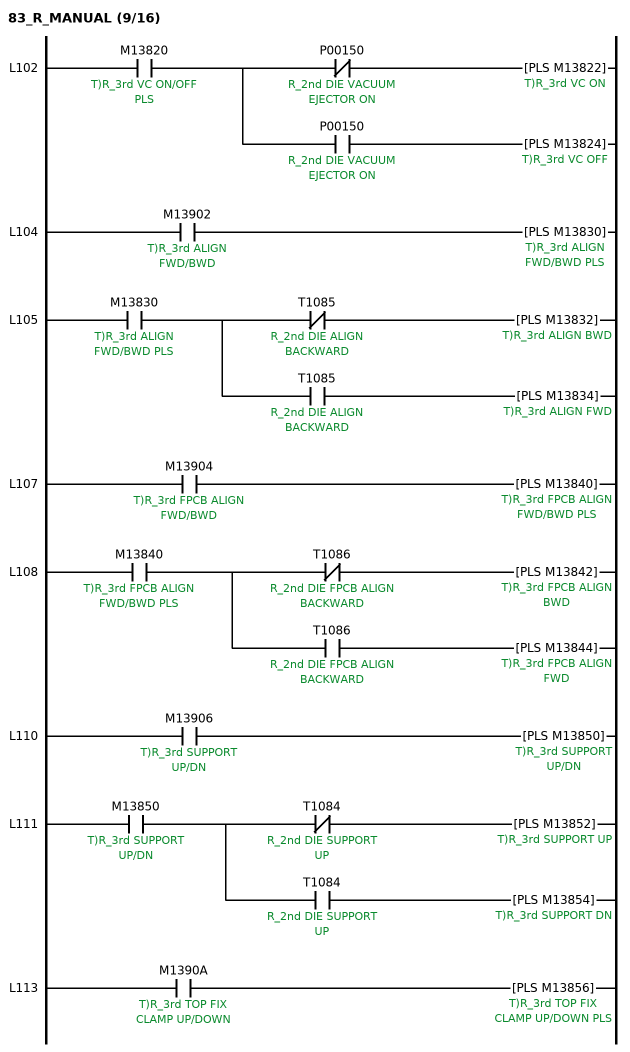
; L102
LOAD      M13820	// T)R_3rd VC ON/OFF PLS
MPUSH
AND NOT   P00150	// R_2nd DIE VACUUM EJECTOR ON
OUTP      M13822	// T)R_3rd VC ON
MPOP
AND       P00150	// R_2nd DIE VACUUM EJECTOR ON
OUTP      M13824	// T)R_3rd VC OFF
; L104
LOAD      M13902	// T)R_3rd ALIGN FWD/BWD
OUTP      M13830	// T)R_3rd ALIGN FWD/BWD PLS
; L105
LOAD      M13830	// T)R_3rd ALIGN FWD/BWD PLS
MPUSH
AND NOT   T1085	// R_2nd DIE ALIGN BACKWARD
OUTP      M13832	// T)R_3rd ALIGN BWD
MPOP
AND       T1085	// R_2nd DIE ALIGN BACKWARD
OUTP      M13834	// T)R_3rd ALIGN FWD
; L107
LOAD      M13904	// T)R_3rd FPCB ALIGN FWD/BWD
OUTP      M13840	// T)R_3rd FPCB ALIGN FWD/BWD PLS
; L108
LOAD      M13840	// T)R_3rd FPCB ALIGN FWD/BWD PLS
MPUSH
AND NOT   T1086	// R_2nd DIE FPCB ALIGN BACKWARD
OUTP      M13842	// T)R_3rd FPCB ALIGN BWD
MPOP
AND       T1086	// R_2nd DIE FPCB ALIGN BACKWARD
OUTP      M13844	// T)R_3rd FPCB ALIGN FWD
; L110
LOAD      M13906	// T)R_3rd SUPPORT UP/DN
OUTP      M13850	// T)R_3rd SUPPORT UP/DN
; L111
LOAD      M13850	// T)R_3rd SUPPORT UP/DN
MPUSH
AND NOT   T1084	// R_2nd DIE SUPPORT UP
OUTP      M13852	// T)R_3rd SUPPORT UP
MPOP
AND       T1084	// R_2nd DIE SUPPORT UP
OUTP      M13854	// T)R_3rd SUPPORT DN
; L113
LOAD      M1390A	// T)R_3rd TOP FIX CLAMP UP/DOWN
OUTP      M13856	// T)R_3rd TOP FIX CLAMP UP/DOWN PLS

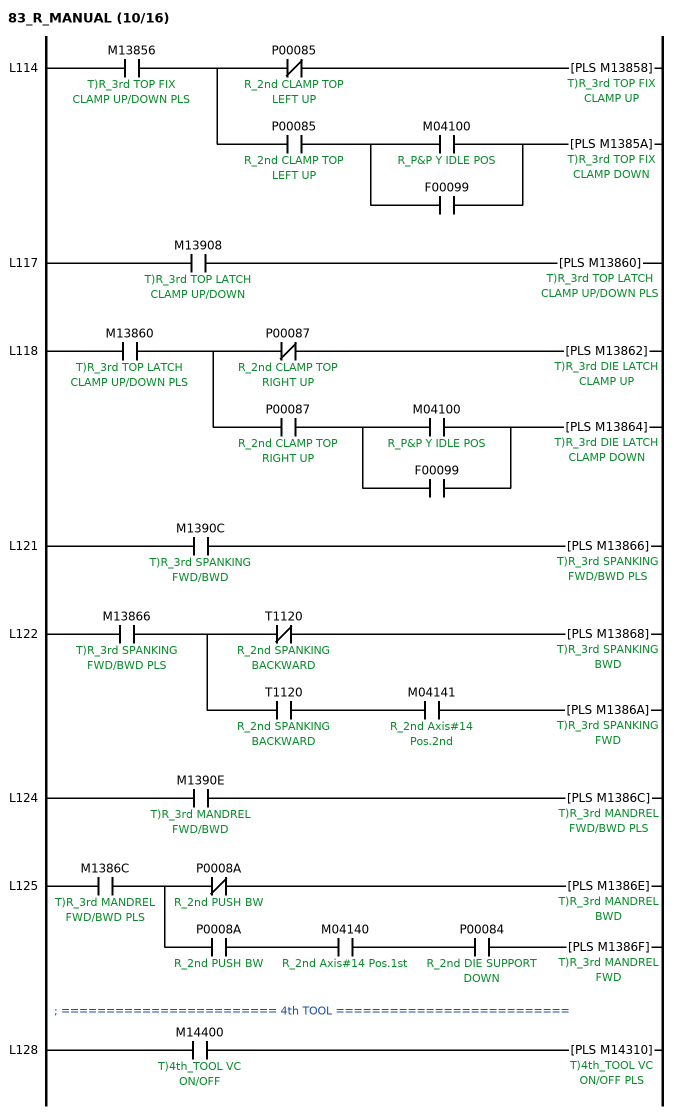
; L114
LOAD      M13856	// T)R_3rd TOP FIX CLAMP UP/DOWN PLS
MPUSH
AND NOT   P00085	// R_2nd CLAMP TOP LEFT UP
OUTP      M13858	// T)R_3rd TOP FIX CLAMP UP
MPOP
AND       P00085	// R_2nd CLAMP TOP LEFT UP
LOAD      M04100	// R_P&P Y IDLE POS
OR        F00099
AND LOAD
OUTP      M1385A	// T)R_3rd TOP FIX CLAMP DOWN
; L117
LOAD      M13908	// T)R_3rd TOP LATCH CLAMP UP/DOWN
OUTP      M13860	// T)R_3rd TOP LATCH CLAMP UP/DOWN PLS
; L118
LOAD      M13860	// T)R_3rd TOP LATCH CLAMP UP/DOWN PLS
MPUSH
AND NOT   P00087	// R_2nd CLAMP TOP RIGHT UP
OUTP      M13862	// T)R_3rd DIE LATCH CLAMP UP
MPOP
AND       P00087	// R_2nd CLAMP TOP RIGHT UP
LOAD      M04100	// R_P&P Y IDLE POS
OR        F00099
AND LOAD
OUTP      M13864	// T)R_3rd DIE LATCH CLAMP DOWN
; L121
LOAD      M1390C	// T)R_3rd SPANKING FWD/BWD
OUTP      M13866	// T)R_3rd SPANKING FWD/BWD PLS
; L122
LOAD      M13866	// T)R_3rd SPANKING FWD/BWD PLS
MPUSH
AND NOT   T1120	// R_2nd SPANKING BACKWARD
OUTP      M13868	// T)R_3rd SPANKING BWD
MPOP
AND       T1120	// R_2nd SPANKING BACKWARD
AND       M04141	// R_2nd Axis#14 Pos.2nd
OUTP      M1386A	// T)R_3rd SPANKING FWD
; L124
LOAD      M1390E	// T)R_3rd MANDREL FWD/BWD
OUTP      M1386C	// T)R_3rd MANDREL FWD/BWD PLS
; L125
LOAD      M1386C	// T)R_3rd MANDREL FWD/BWD PLS
MPUSH
AND NOT   P0008A	// R_2nd PUSH BW
OUTP      M1386E	// T)R_3rd MANDREL BWD
MPOP
AND       P0008A	// R_2nd PUSH BW
AND       M04140	// R_2nd Axis#14 Pos.1st
AND       P00084	// R_2nd DIE SUPPORT DOWN
OUTP      M1386F	// T)R_3rd MANDREL FWD
// ======================== 4th TOOL ==========================
; L128
LOAD      M14400	// T)4th_TOOL VC ON/OFF
OUTP      M14310	// T)4th_TOOL VC ON/OFF PLS

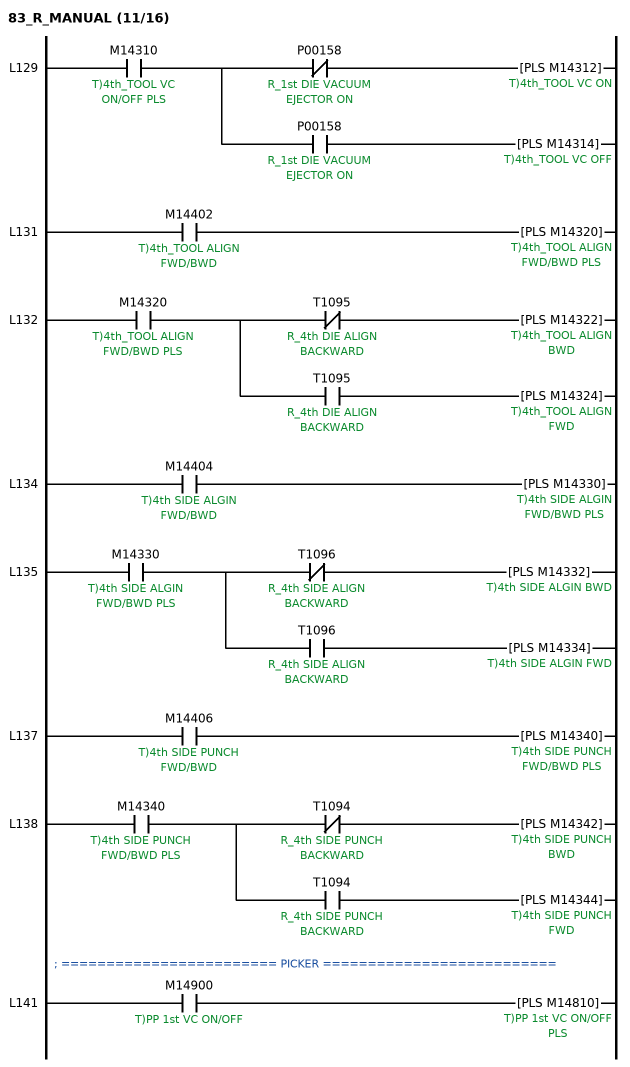
; L129
LOAD      M14310	// T)4th_TOOL VC ON/OFF PLS
MPUSH
AND NOT   P00158	// R_1st DIE VACUUM EJECTOR ON
OUTP      M14312	// T)4th_TOOL VC ON
MPOP
AND       P00158	// R_1st DIE VACUUM EJECTOR ON
OUTP      M14314	// T)4th_TOOL VC OFF
; L131
LOAD      M14402	// T)4th_TOOL ALIGN FWD/BWD
OUTP      M14320	// T)4th_TOOL ALIGN FWD/BWD PLS
; L132
LOAD      M14320	// T)4th_TOOL ALIGN FWD/BWD PLS
MPUSH
AND NOT   T1095	// R_4th DIE ALIGN BACKWARD
OUTP      M14322	// T)4th_TOOL ALIGN BWD
MPOP
AND       T1095	// R_4th DIE ALIGN BACKWARD
OUTP      M14324	// T)4th_TOOL ALIGN FWD
; L134
LOAD      M14404	// T)4th SIDE ALGIN FWD/BWD
OUTP      M14330	// T)4th SIDE ALGIN FWD/BWD PLS
; L135
LOAD      M14330	// T)4th SIDE ALGIN FWD/BWD PLS
MPUSH
AND NOT   T1096	// R_4th SIDE ALIGN BACKWARD
OUTP      M14332	// T)4th SIDE ALGIN BWD
MPOP
AND       T1096	// R_4th SIDE ALIGN BACKWARD
OUTP      M14334	// T)4th SIDE ALGIN FWD
; L137
LOAD      M14406	// T)4th SIDE PUNCH FWD/BWD
OUTP      M14340	// T)4th SIDE PUNCH FWD/BWD PLS
; L138
LOAD      M14340	// T)4th SIDE PUNCH FWD/BWD PLS
MPUSH
AND NOT   T1094	// R_4th SIDE PUNCH BACKWARD
OUTP      M14342	// T)4th SIDE PUNCH BWD
MPOP
AND       T1094	// R_4th SIDE PUNCH BACKWARD
OUTP      M14344	// T)4th SIDE PUNCH FWD
// ======================== PICKER ==========================
; L141
LOAD      M14900	// T)PP 1st VC ON/OFF
OUTP      M14810	// T)PP 1st VC ON/OFF PLS

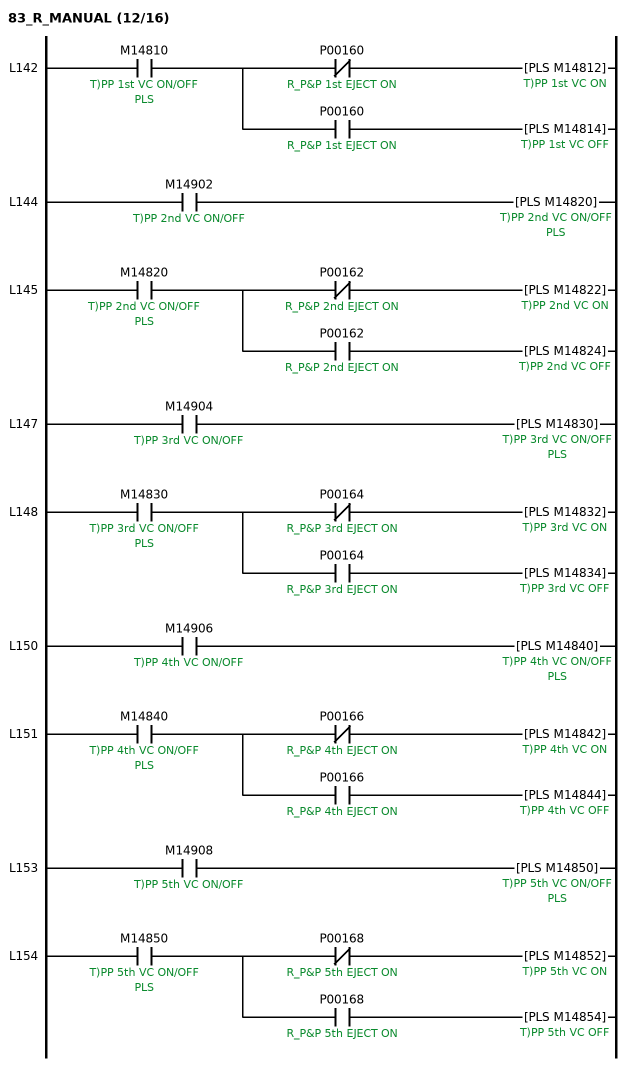
; L142
LOAD      M14810	// T)PP 1st VC ON/OFF PLS
MPUSH
AND NOT   P00160	// R_P&P 1st EJECT ON
OUTP      M14812	// T)PP 1st VC ON
MPOP
AND       P00160	// R_P&P 1st EJECT ON
OUTP      M14814	// T)PP 1st VC OFF
; L144
LOAD      M14902	// T)PP 2nd VC ON/OFF
OUTP      M14820	// T)PP 2nd VC ON/OFF PLS
; L145
LOAD      M14820	// T)PP 2nd VC ON/OFF PLS
MPUSH
AND NOT   P00162	// R_P&P 2nd EJECT ON
OUTP      M14822	// T)PP 2nd VC ON
MPOP
AND       P00162	// R_P&P 2nd EJECT ON
OUTP      M14824	// T)PP 2nd VC OFF
; L147
LOAD      M14904	// T)PP 3rd VC ON/OFF
OUTP      M14830	// T)PP 3rd VC ON/OFF PLS
; L148
LOAD      M14830	// T)PP 3rd VC ON/OFF PLS
MPUSH
AND NOT   P00164	// R_P&P 3rd EJECT ON
OUTP      M14832	// T)PP 3rd VC ON
MPOP
AND       P00164	// R_P&P 3rd EJECT ON
OUTP      M14834	// T)PP 3rd VC OFF
; L150
LOAD      M14906	// T)PP 4th VC ON/OFF
OUTP      M14840	// T)PP 4th VC ON/OFF PLS
; L151
LOAD      M14840	// T)PP 4th VC ON/OFF PLS
MPUSH
AND NOT   P00166	// R_P&P 4th EJECT ON
OUTP      M14842	// T)PP 4th VC ON
MPOP
AND       P00166	// R_P&P 4th EJECT ON
OUTP      M14844	// T)PP 4th VC OFF
; L153
LOAD      M14908	// T)PP 5th VC ON/OFF
OUTP      M14850	// T)PP 5th VC ON/OFF PLS
; L154
LOAD      M14850	// T)PP 5th VC ON/OFF PLS
MPUSH
AND NOT   P00168	// R_P&P 5th EJECT ON
OUTP      M14852	// T)PP 5th VC ON
MPOP
AND       P00168	// R_P&P 5th EJECT ON
OUTP      M14854	// T)PP 5th VC OFF

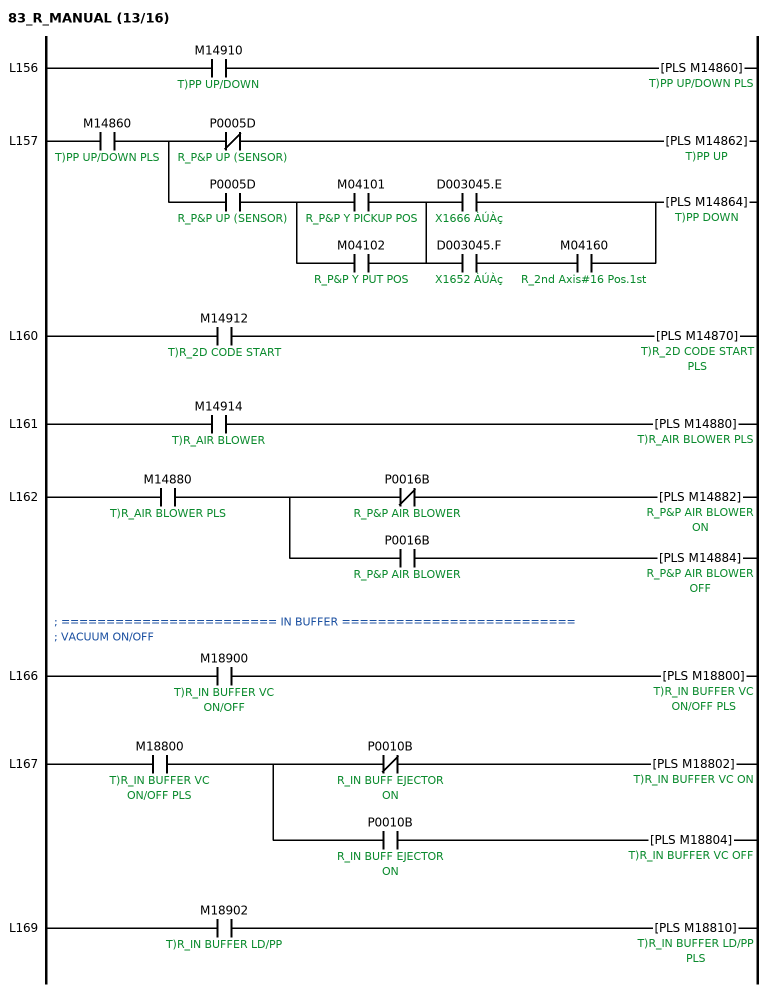
; L156
LOAD      M14910	// T)PP UP/DOWN
OUTP      M14860	// T)PP UP/DOWN PLS
; L157
LOAD      M14860	// T)PP UP/DOWN PLS
MPUSH
AND NOT   P0005D	// R_P&P UP (SENSOR)
OUTP      M14862	// T)PP UP
MPOP
AND       P0005D	// R_P&P UP (SENSOR)
LOAD      M04101	// R_P&P Y PICKUP POS
OR        M04102	// R_P&P Y PUT POS
AND LOAD
LOAD      D003045.E	// X1666 ÀÚÀç
LOAD      D003045.F	// X1652 ÀÚÀç
AND       M04160	// R_2nd Axis#16 Pos.1st
OR LOAD
AND LOAD
OUTP      M14864	// T)PP DOWN
; L160
LOAD      M14912	// T)R_2D CODE START
OUTP      M14870	// T)R_2D CODE START PLS
; L161
LOAD      M14914	// T)R_AIR BLOWER
OUTP      M14880	// T)R_AIR BLOWER PLS
; L162
LOAD      M14880	// T)R_AIR BLOWER PLS
MPUSH
AND NOT   P0016B	// R_P&P AIR BLOWER
OUTP      M14882	// R_P&P AIR BLOWER ON
MPOP
AND       P0016B	// R_P&P AIR BLOWER
OUTP      M14884	// R_P&P AIR BLOWER OFF
// ======================== IN BUFFER ==========================
// VACUUM ON/OFF
; L166
LOAD      M18900	// T)R_IN BUFFER VC ON/OFF
OUTP      M18800	// T)R_IN BUFFER VC ON/OFF PLS
; L167
LOAD      M18800	// T)R_IN BUFFER VC ON/OFF PLS
MPUSH
AND NOT   P0010B	// R_IN BUFF EJECTOR ON
OUTP      M18802	// T)R_IN BUFFER VC ON
MPOP
AND       P0010B	// R_IN BUFF EJECTOR ON
OUTP      M18804	// T)R_IN BUFFER VC OFF
; L169
LOAD      M18902	// T)R_IN BUFFER LD/PP
OUTP      M18810	// T)R_IN BUFFER LD/PP PLS

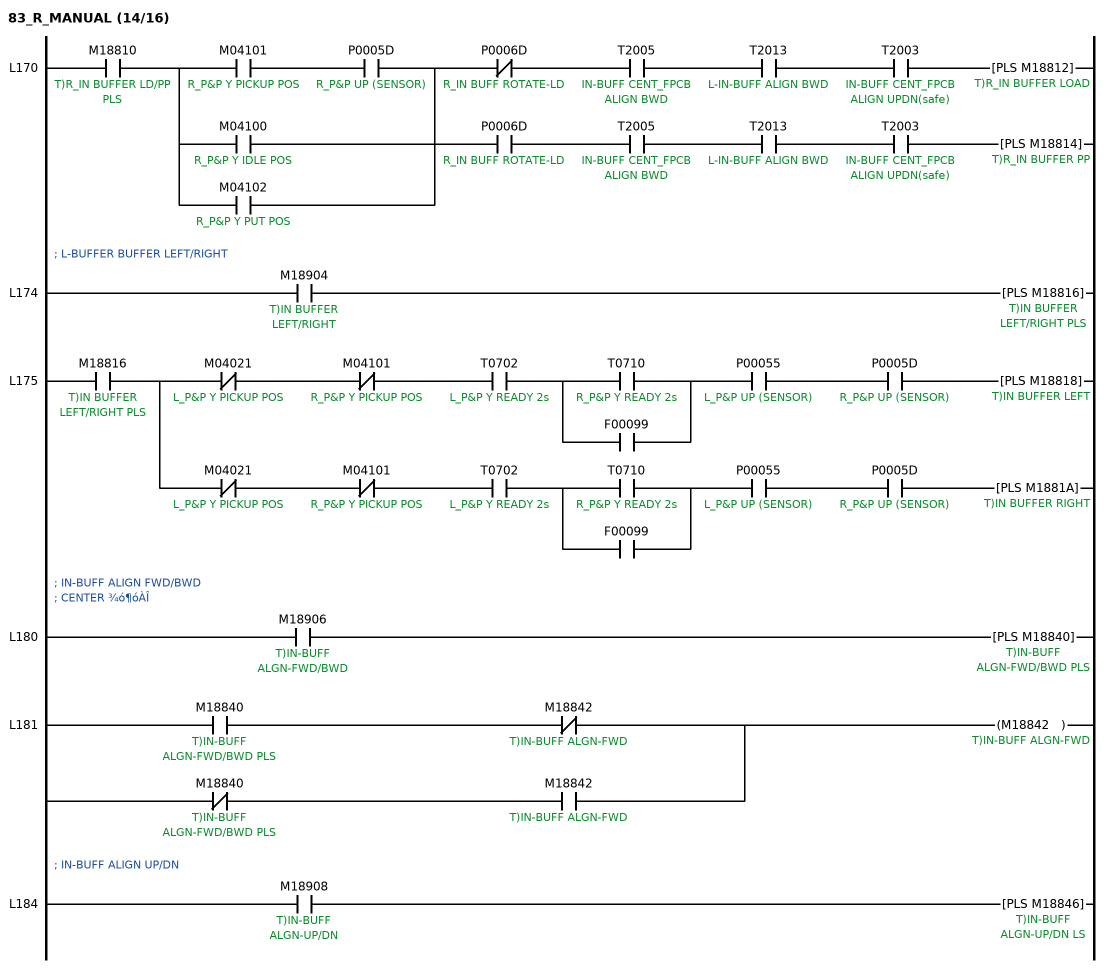
; L170
LOAD      M18810	// T)R_IN BUFFER LD/PP PLS
LOAD      M04101	// R_P&P Y PICKUP POS
AND       P0005D	// R_P&P UP (SENSOR)
OR        M04100	// R_P&P Y IDLE POS
OR        M04102	// R_P&P Y PUT POS
AND LOAD
MPUSH
AND NOT   P0006D	// R_IN BUFF ROTATE-LD
AND       T2005	// IN-BUFF CENT_FPCB ALIGN BWD
AND       T2013	// L-IN-BUFF ALIGN BWD
AND       T2003	// IN-BUFF CENT_FPCB ALIGN UPDN(safe)
OUTP      M18812	// T)R_IN BUFFER LOAD
MPOP
AND       P0006D	// R_IN BUFF ROTATE-LD
AND       T2005	// IN-BUFF CENT_FPCB ALIGN BWD
AND       T2013	// L-IN-BUFF ALIGN BWD
AND       T2003	// IN-BUFF CENT_FPCB ALIGN UPDN(safe)
OUTP      M18814	// T)R_IN BUFFER PP
// L-BUFFER BUFFER LEFT/RIGHT
; L174
LOAD      M18904	// T)IN BUFFER LEFT/RIGHT
OUTP      M18816	// T)IN BUFFER LEFT/RIGHT PLS
; L175
LOAD      M18816	// T)IN BUFFER LEFT/RIGHT PLS
MPUSH
AND NOT   M04021	// L_P&P Y PICKUP POS
AND NOT   M04101	// R_P&P Y PICKUP POS
AND       T0702	// L_P&P Y READY 2s
LOAD      T0710	// R_P&P Y READY 2s
OR        F00099
AND LOAD
AND       P00055	// L_P&P UP (SENSOR)
AND       P0005D	// R_P&P UP (SENSOR)
OUTP      M18818	// T)IN BUFFER LEFT
MPOP
AND NOT   M04021	// L_P&P Y PICKUP POS
AND NOT   M04101	// R_P&P Y PICKUP POS
AND       T0702	// L_P&P Y READY 2s
LOAD      T0710	// R_P&P Y READY 2s
OR        F00099
AND LOAD
AND       P00055	// L_P&P UP (SENSOR)
AND       P0005D	// R_P&P UP (SENSOR)
OUTP      M1881A	// T)IN BUFFER RIGHT
// IN-BUFF ALIGN FWD/BWD
; L180
LOAD      M18906	// T)IN-BUFF ALGN-FWD/BWD
OUTP      M18840	// T)IN-BUFF ALGN-FWD/BWD PLS
// output comment: CENTER ¾ó¶óÀÎ
; L181
LOAD      M18840	// T)IN-BUFF ALGN-FWD/BWD PLS
AND NOT   M18842	// T)IN-BUFF ALGN-FWD
LOAD NOT  M18840	// T)IN-BUFF ALGN-FWD/BWD PLS
AND       M18842	// T)IN-BUFF ALGN-FWD
OR LOAD
OUT       M18842	// T)IN-BUFF ALGN-FWD
// IN-BUFF ALIGN UP/DN
; L184
LOAD      M18908	// T)IN-BUFF ALGN-UP/DN
OUTP      M18846	// T)IN-BUFF ALGN-UP/DN LS

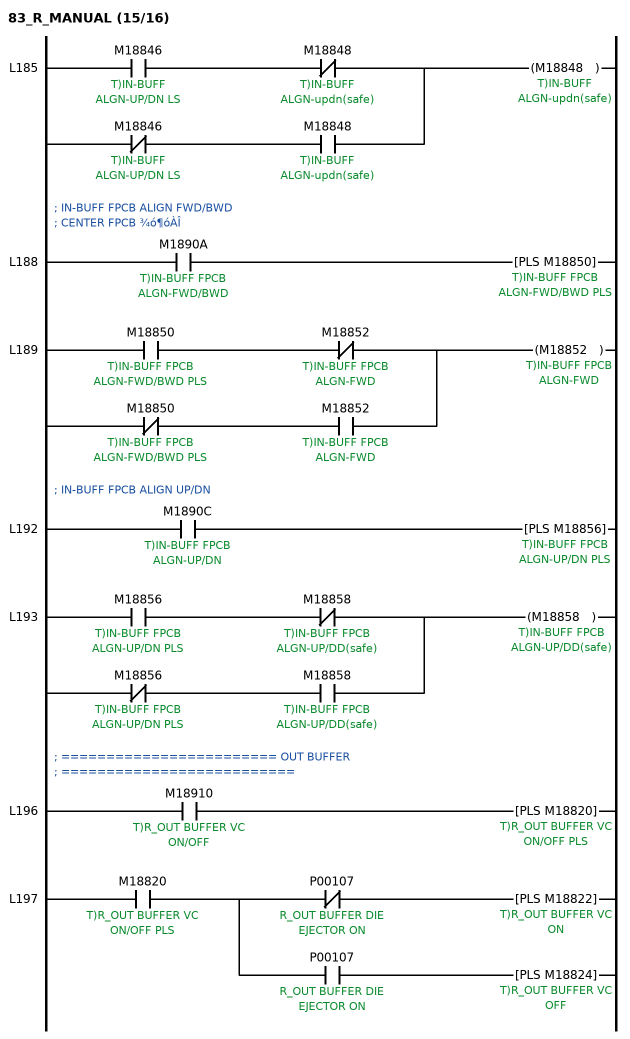
; L185
LOAD      M18846	// T)IN-BUFF ALGN-UP/DN LS
AND NOT   M18848	// T)IN-BUFF ALGN-updn(safe)
LOAD NOT  M18846	// T)IN-BUFF ALGN-UP/DN LS
AND       M18848	// T)IN-BUFF ALGN-updn(safe)
OR LOAD
OUT       M18848	// T)IN-BUFF ALGN-updn(safe)
// IN-BUFF FPCB ALIGN FWD/BWD
; L188
LOAD      M1890A	// T)IN-BUFF FPCB ALGN-FWD/BWD
OUTP      M18850	// T)IN-BUFF FPCB ALGN-FWD/BWD PLS
// output comment: CENTER FPCB ¾ó¶óÀÎ
; L189
LOAD      M18850	// T)IN-BUFF FPCB ALGN-FWD/BWD PLS
AND NOT   M18852	// T)IN-BUFF FPCB ALGN-FWD
LOAD NOT  M18850	// T)IN-BUFF FPCB ALGN-FWD/BWD PLS
AND       M18852	// T)IN-BUFF FPCB ALGN-FWD
OR LOAD
OUT       M18852	// T)IN-BUFF FPCB ALGN-FWD
// IN-BUFF FPCB ALIGN UP/DN
; L192
LOAD      M1890C	// T)IN-BUFF FPCB ALGN-UP/DN
OUTP      M18856	// T)IN-BUFF FPCB ALGN-UP/DN PLS
; L193
LOAD      M18856	// T)IN-BUFF FPCB ALGN-UP/DN PLS
AND NOT   M18858	// T)IN-BUFF FPCB ALGN-UP/DD(safe)
LOAD NOT  M18856	// T)IN-BUFF FPCB ALGN-UP/DN PLS
AND       M18858	// T)IN-BUFF FPCB ALGN-UP/DD(safe)
OR LOAD
OUT       M18858	// T)IN-BUFF FPCB ALGN-UP/DD(safe)
// ======================== OUT BUFFER ==========================
; L196
LOAD      M18910	// T)R_OUT BUFFER VC ON/OFF
OUTP      M18820	// T)R_OUT BUFFER VC ON/OFF PLS
; L197
LOAD      M18820	// T)R_OUT BUFFER VC ON/OFF PLS
MPUSH
AND NOT   P00107	// R_OUT BUFFER DIE EJECTOR ON
OUTP      M18822	// T)R_OUT BUFFER VC ON
MPOP
AND       P00107	// R_OUT BUFFER DIE EJECTOR ON
OUTP      M18824	// T)R_OUT BUFFER VC OFF

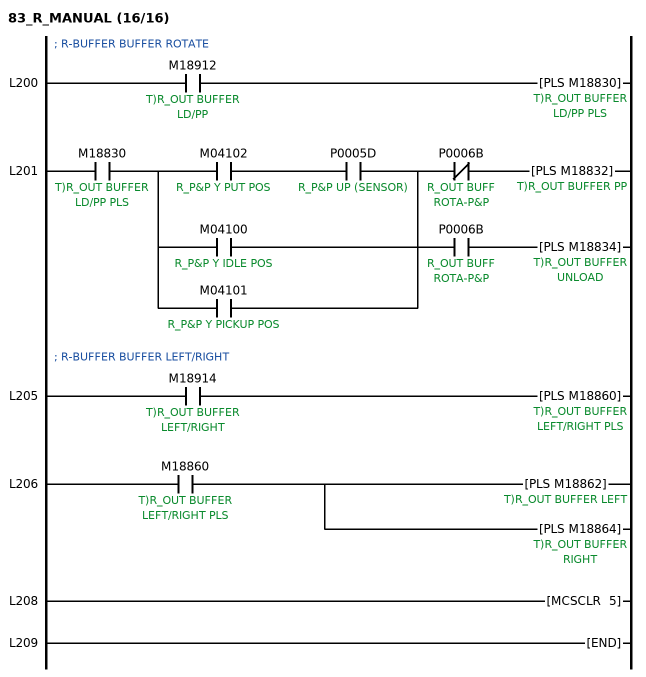
// R-BUFFER BUFFER ROTATE
; L200
LOAD      M18912	// T)R_OUT BUFFER LD/PP
OUTP      M18830	// T)R_OUT BUFFER LD/PP PLS
; L201
LOAD      M18830	// T)R_OUT BUFFER LD/PP PLS
LOAD      M04102	// R_P&P Y PUT POS
AND       P0005D	// R_P&P UP (SENSOR)
OR        M04100	// R_P&P Y IDLE POS
OR        M04101	// R_P&P Y PICKUP POS
AND LOAD
MPUSH
AND NOT   P0006B	// R_OUT BUFF ROTA-P&P
OUTP      M18832	// T)R_OUT BUFFER PP
MPOP
AND       P0006B	// R_OUT BUFF ROTA-P&P
OUTP      M18834	// T)R_OUT BUFFER UNLOAD
// R-BUFFER BUFFER LEFT/RIGHT
; L205
LOAD      M18914	// T)R_OUT BUFFER LEFT/RIGHT
OUTP      M18860	// T)R_OUT BUFFER LEFT/RIGHT PLS
; L206
LOAD      M18860	// T)R_OUT BUFFER LEFT/RIGHT PLS
OUTP      M18862	// T)R_OUT BUFFER LEFT
OUTP      M18864	// T)R_OUT BUFFER RIGHT
; L208
MCSCLR    5
; L209
END

PROGRAM 84_RUN_TIME (task: ½ºÄµ ÇÁ·Î±×·¥)

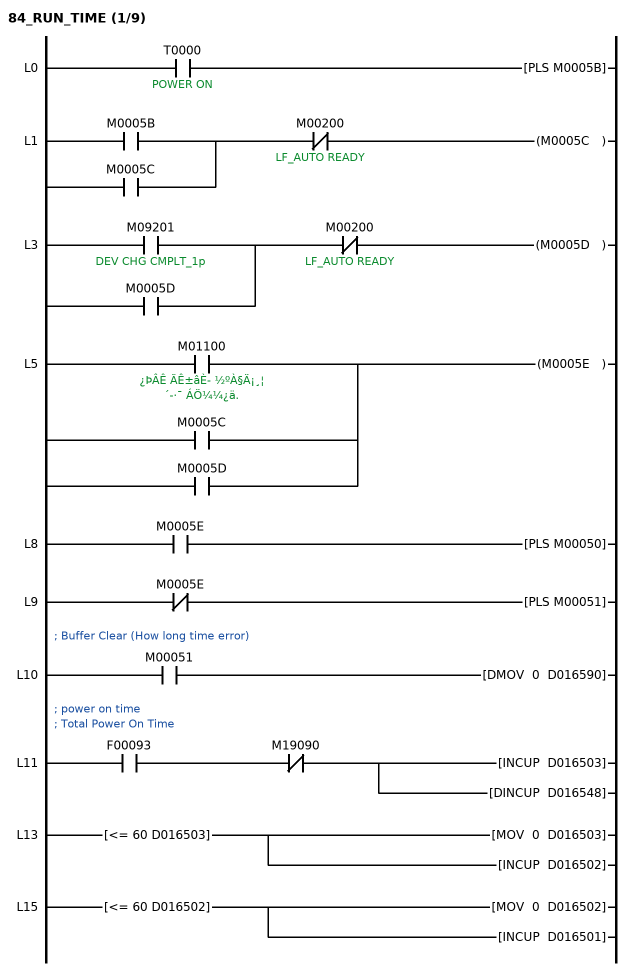
; L0
LOAD      T0000	// POWER ON
OUTP      M0005B
; L1
LOAD      M0005B
OR        M0005C
AND NOT   M00200	// LF_AUTO READY
OUT       M0005C
; L3
LOAD      M09201	// DEV CHG CMPLT_1p
OR        M0005D
AND NOT   M00200	// LF_AUTO READY
OUT       M0005D
; L5
LOAD      M01100	// ¿ÞÂÊ ÃÊ±âÈ­ ½ºÀ§Ä¡¸¦ ´­·¯ ÁÖ¼¼¿ä.
OR        M0005C
OR        M0005D
OUT       M0005E
; L8
LOAD      M0005E
OUTP      M00050
; L9
LOAD NOT  M0005E
OUTP      M00051
; L10
LOAD      M00051
DMOV      0 D016590
// output comment: Buffer Clear (How long time error)
; L11
LOAD      F00093
AND NOT   M19090
INCUP     D016503
DINCUP    D016548
// output comment: power on time
// output comment: Total Power On Time
; L13
LOAD<=    60 D016503
MOV       0 D016503
INCUP     D016502
; L15
LOAD<=    60 D016502
MOV       0 D016502
INCUP     D016501

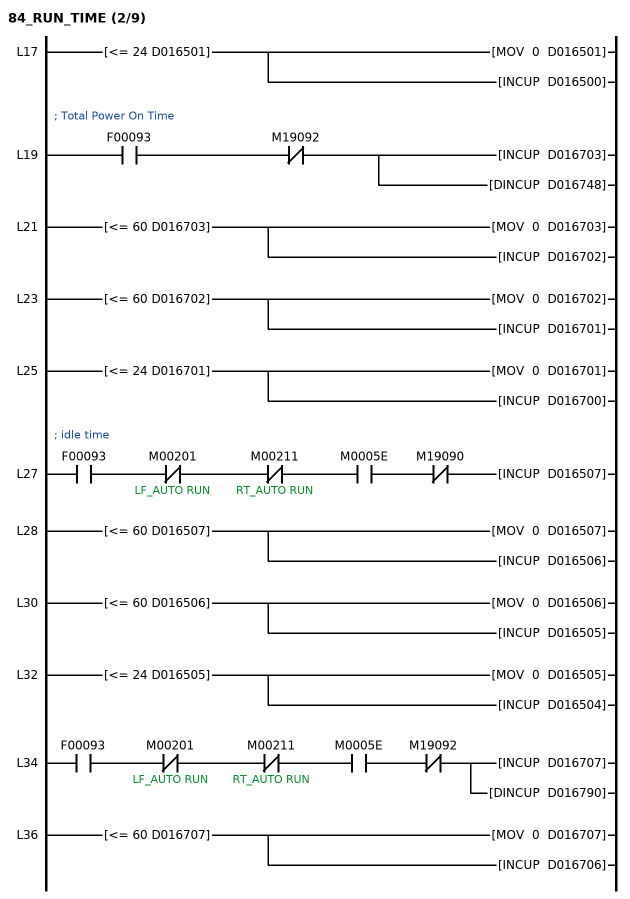
; L17
LOAD<=    24 D016501
MOV       0 D016501
INCUP     D016500
; L19
LOAD      F00093
AND NOT   M19092
INCUP     D016703
DINCUP    D016748
// output comment: Total Power On Time
; L21
LOAD<=    60 D016703
MOV       0 D016703
INCUP     D016702
; L23
LOAD<=    60 D016702
MOV       0 D016702
INCUP     D016701
; L25
LOAD<=    24 D016701
MOV       0 D016701
INCUP     D016700
; L27
LOAD      F00093
AND NOT   M00201	// LF_AUTO RUN
AND NOT   M00211	// RT_AUTO RUN
AND       M0005E
AND NOT   M19090
INCUP     D016507
// output comment: idle time
; L28
LOAD<=    60 D016507
MOV       0 D016507
INCUP     D016506
; L30
LOAD<=    60 D016506
MOV       0 D016506
INCUP     D016505
; L32
LOAD<=    24 D016505
MOV       0 D016505
INCUP     D016504
; L34
LOAD      F00093
AND NOT   M00201	// LF_AUTO RUN
AND NOT   M00211	// RT_AUTO RUN
AND       M0005E
AND NOT   M19092
INCUP     D016707
DINCUP    D016790
; L36
LOAD<=    60 D016707
MOV       0 D016707
INCUP     D016706

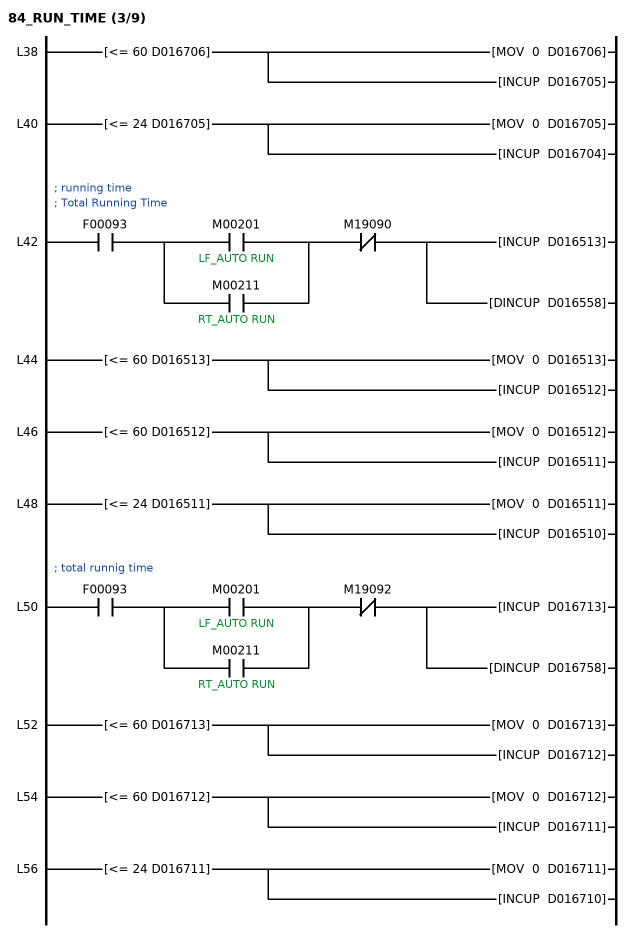
; L38
LOAD<=    60 D016706
MOV       0 D016706
INCUP     D016705
; L40
LOAD<=    24 D016705
MOV       0 D016705
INCUP     D016704
; L42
LOAD      F00093
LOAD      M00201	// LF_AUTO RUN
OR        M00211	// RT_AUTO RUN
AND LOAD
AND NOT   M19090
INCUP     D016513
DINCUP    D016558
// output comment: running time
// output comment: Total Running Time
; L44
LOAD<=    60 D016513
MOV       0 D016513
INCUP     D016512
; L46
LOAD<=    60 D016512
MOV       0 D016512
INCUP     D016511
; L48
LOAD<=    24 D016511
MOV       0 D016511
INCUP     D016510
; L50
LOAD      F00093
LOAD      M00201	// LF_AUTO RUN
OR        M00211	// RT_AUTO RUN
AND LOAD
AND NOT   M19092
INCUP     D016713
DINCUP    D016758
// output comment: total runnig time
; L52
LOAD<=    60 D016713
MOV       0 D016713
INCUP     D016712
; L54
LOAD<=    60 D016712
MOV       0 D016712
INCUP     D016711
; L56
LOAD<=    24 D016711
MOV       0 D016711
INCUP     D016710

